C03649=1235.303,242.805,-59.932,-176.879,6.176,148.185
C03650=1235.299,243.053,-59.959,-176.877,6.178,148.185
C03651=1235.294,243.302,-59.985,-176.875,6.180,148.185
C03652=1235.290,243.551,-60.011,-176.872,6.182,148.184
C03653=1235.286,243.800,-60.036,-176.870,6.184,148.184
C03654=1235.281,244.047,-60.063,-176.867,6.186,148.184
C03655=1235.276,244.296,-60.089,-176.864,6.187,148.184
C03656=1235.272,244.545,-60.115,-176.862,6.189,148.183
C03657=1235.268,244.793,-60.141,-176.860,6.191,148.183
C03658=1235.263,245.043,-60.167,-176.858,6.193,148.183
C03659=1235.259,245.291,-60.193,-176.855,6.195,148.183
C03660=1235.254,245.539,-60.220,-176.852,6.196,148.182
C03661=1235.249,245.788,-60.246,-176.850,6.198,148.182
C03662=1235.246,246.036,-60.272,-176.847,6.200,148.182
C03663=1235.241,246.285,-60.298,-176.844,6.202,148.181
C03664=1235.236,246.534,-60.324,-176.842,6.204,148.181
C03665=1235.232,246.783,-60.351,-176.840,6.206,148.181
C03666=1235.227,247.031,-60.377,-176.837,6.208,148.181
C03667=1235.224,247.280,-60.404,-176.835,6.210,148.180
C03668=1235.218,247.528,-60.429,-176.832,6.211,148.180
C03669=1235.214,247.776,-60.456,-176.830,6.213,148.180
C03670=1235.209,248.025,-60.482,-176.828,6.215,148.180
C03671=1235.205,248.273,-60.509,-176.825,6.217,148.179
C03672=1235.200,248.523,-60.535,-176.823,6.219,148.179
C03673=1235.196,248.771,-60.562,-176.820,6.221,148.179
C03674=1235.192,249.020,-60.587,-176.817,6.223,148.178
C03675=1235.187,249.268,-60.614,-176.815,6.225,148.178
C03676=1235.183,249.517,-60.640,-176.813,6.227,148.178
C03677=1235.179,249.765,-60.667,-176.810,6.229,148.178
C03678=1235.175,250.013,-60.694,-176.807,6.231,148.177
C03679=1235.170,250.263,-60.720,-176.805,6.232,148.177
C03680=1235.166,250.511,-60.746,-176.802,6.234,148.177
C03681=1235.160,250.759,-60.772,-176.800,6.237,148.177
C03682=1235.156,251.007,-60.799,-176.797,6.238,148.176
C03683=1235.152,251.256,-60.826,-176.795,6.240,148.176
C03684=1235.147,251.505,-60.852,-176.793,6.241,148.176
C03685=1235.143,251.753,-60.879,-176.790,6.243,148.175
C03686=1235.138,252.002,-60.905,-176.788,6.245,148.175
C03687=1235.134,252.250,-60.932,-176.785,6.247,148.175
C03688=1235.129,252.499,-60.959,-176.783,6.249,148.175
C03689=1235.125,252.747,-60.985,-176.780,6.251,148.174
C03690=1235.120,252.996,-61.011,-176.778,6.253,148.174
C03691=1235.116,253.245,-61.039,-176.776,6.255,148.174
C03692=1235.112,253.493,-61.065,-176.773,6.257,148.174
C03693=1235.107,253.742,-61.091,-176.770,6.259,148.173
C03694=1235.103,253.990,-61.118,-176.768,6.261,148.173
C03695=1235.098,254.239,-61.145,-176.766,6.263,148.173
C03696=1235.093,254.487,-61.172,-176.763,6.265,148.173
C03697=1235.089,254.736,-61.198,-176.760,6.267,148.172
C03698=1235.085,254.985,-61.225,-176.758,6.269,148.172
C03699=1235.080,255.233,-61.252,-176.755,6.271,148.172
C03700=1235.076,255.481,-61.278,-176.753,6.273,148.172
C03701=1235.071,255.730,-61.305,-176.750,6.275,148.171
C03702=1235.067,255.978,-61.332,-176.748,6.277,148.171
C03703=1235.062,256.227,-61.358,-176.745,6.279,148.171
C03704=1235.058,256.476,-61.386,-176.743,6.281,148.171
C03705=1235.054,256.725,-61.413,-176.741,6.283,148.170
C03706=1235.050,256.973,-61.439,-176.738,6.285,148.170
C03707=1235.045,257.221,-61.466,-176.735,6.287,148.170
C03708=1235.041,257.470,-61.493,-176.733,6.289,148.170
C03709=1235.037,257.718,-61.520,-176.731,6.291,148.169
C03710=1235.032,257.967,-61.547,-176.728,6.293,148.169
C03711=1235.027,258.216,-61.573,-176.726,6.295,148.169
C03712=1235.022,258.464,-61.600,-176.723,6.297,148.169
C03713=1235.018,258.712,-61.627,-176.721,6.299,148.168
C03714=1235.014,258.961,-61.654,-176.718,6.300,148.168
C03715=1235.009,259.209,-61.681,-176.716,6.303,148.168
C03716=1235.004,259.458,-61.708,-176.713,6.305,148.168
C03717=1235.001,259.707,-61.735,-176.711,6.306,148.167
C03718=1234.996,259.955,-61.762,-176.708,6.308,148.167
C03719=1234.992,260.204,-61.789,-176.706,6.311,148.167
C03720=1234.987,260.452,-61.816,-176.703,6.312,148.167
C03721=1234.983,260.701,-61.843,-176.701,6.314,148.166
C03722=1234.979,260.949,-61.869,-176.699,6.317,148.166
C03723=1234.974,261.197,-61.897,-176.696,6.318,148.166
C03724=1234.970,261.445,-61.924,-176.694,6.320,148.166
C03725=1234.966,261.694,-61.952,-176.691,6.322,148.165
C03726=1234.961,261.943,-61.979,-176.689,6.324,148.165
C03727=1234.956,262.191,-62.006,-176.686,6.326,148.165
C03728=1234.952,262.440,-62.032,-176.684,6.328,148.165
C03729=1234.948,262.688,-62.059,-176.681,6.330,148.165
C03730=1234.943,262.937,-62.086,-176.679,6.332,148.164
C03731=1234.939,263.186,-62.114,-176.676,6.334,148.164
C03732=1234.934,263.458,-62.143,-176.674,6.336,148.164
C03733=1234.929,263.731,-62.174,-176.672,6.338,148.164
C03734=1234.925,264.003,-62.204,-176.668,6.341,148.163
C03735=1234.919,264.276,-62.234,-176.666,6.343,148.163
C03736=1234.915,264.524,-62.261,-176.663,6.345,148.163
C03737=1234.911,264.772,-62.287,-176.661,6.347,148.163
C03738=1234.906,265.021,-62.314,-176.659,6.349,148.162
C03739=1234.902,265.269,-62.343,-176.656,6.351,148.162
C03740=1234.898,265.518,-62.370,-176.654,6.353,148.162
C03741=1234.893,265.766,-62.397,-176.651,6.355,148.162
C03742=1234.888,266.015,-62.424,-176.649,6.357,148.161
C03743=1234.884,266.263,-62.452,-176.646,6.359,148.161
C03744=1234.880,266.512,-62.479,-176.644,6.361,148.161
C03745=1234.875,266.761,-62.506,-176.641,6.363,148.161
C03746=1234.871,267.009,-62.533,-176.639,6.365,148.161
C03747=1234.866,267.257,-62.561,-176.637,6.367,148.160
C03748=1234.862,267.506,-62.588,-176.634,6.369,148.160
C03749=1234.858,267.754,-62.616,-176.632,6.371,148.160
C03750=1234.853,268.002,-62.643,-176.629,6.373,148.160
C03751=1234.849,268.251,-62.670,-176.627,6.375,148.160
C03752=1234.845,268.500,-62.698,-176.625,6.377,148.159
C03753=1234.840,268.748,-62.725,-176.622,6.379,148.159
C03754=1234.836,268.997,-62.752,-176.619,6.382,148.159
C03755=1234.831,269.244,-62.780,-176.617,6.384,148.159
C03756=1234.827,269.494,-62.808,-176.614,6.386,148.159
C03757=1234.823,269.741,-62.835,-176.612,6.388,148.158
C03758=1234.817,269.990,-62.863,-176.609,6.390,148.158
C03759=1234.814,270.239,-62.891,-176.607,6.392,148.158
C03760=1234.809,270.487,-62.918,-176.605,6.394,148.158
C03761=1234.805,270.735,-62.946,-176.602,6.396,148.157
C03762=1234.800,270.984,-62.973,-176.600,6.398,148.157
C03763=1234.796,271.232,-63.001,-176.597,6.400,148.157
C03764=1234.792,271.481,-63.028,-176.595,6.402,148.157
C03765=1234.787,271.729,-63.056,-176.593,6.404,148.157
C03766=1234.783,271.978,-63.084,-176.590,6.406,148.156
C03767=1234.778,272.226,-63.112,-176.588,6.408,148.156
C03768=1234.773,272.475,-63.139,-176.585,6.410,148.156
C03769=1234.770,272.723,-63.167,-176.583,6.413,148.156
C03770=1234.765,272.972,-63.194,-176.581,6.414,148.156
C03771=1234.761,273.219,-63.222,-176.578,6.418,148.156
C03772=1234.757,273.468,-63.250,-176.575,6.419,148.155
C03773=1234.752,273.717,-63.278,-176.573,6.421,148.155
C03774=1234.747,273.965,-63.306,-176.571,6.424,148.155
C03775=1234.743,274.214,-63.333,-176.568,6.425,148.155
C03776=1234.739,274.462,-63.361,-176.566,6.428,148.155
C03777=1234.735,274.710,-63.389,-176.563,6.430,148.154
C03778=1234.730,274.959,-63.417,-176.561,6.432,148.154
C03779=1234.725,275.207,-63.444,-176.559,6.434,148.154
C03780=1234.722,275.456,-63.472,-176.556,6.436,148.154
C03781=1234.717,275.704,-63.500,-176.554,6.438,148.154
C03782=1234.712,275.952,-63.528,-176.551,6.440,148.153
C03783=1234.708,276.201,-63.556,-176.549,6.442,148.153
C03784=1234.704,276.449,-63.584,-176.546,6.445,148.153
C03785=1234.700,276.698,-63.611,-176.544,6.447,148.153
C03786=1234.695,276.946,-63.640,-176.541,6.449,148.153
C03787=1234.690,277.194,-63.667,-176.539,6.451,148.153
C03788=1234.686,277.443,-63.696,-176.537,6.453,148.152
C03789=1234.682,277.690,-63.723,-176.535,6.455,148.152
C03790=1234.677,277.940,-63.751,-176.532,6.457,148.152
C03791=1234.673,278.188,-63.779,-176.530,6.459,148.152
C03792=1234.669,278.436,-63.807,-176.527,6.461,148.152
C03793=1234.664,278.685,-63.836,-176.525,6.463,148.152
C03794=1234.660,278.933,-63.864,-176.523,6.465,148.151
C03795=1234.656,279.181,-63.892,-176.520,6.468,148.151
C03796=1234.651,279.430,-63.919,-176.517,6.470,148.151
C03797=1234.647,279.678,-63.947,-176.515,6.473,148.151
C03798=1234.642,279.927,-63.976,-176.513,6.474,148.151
C03799=1234.638,280.175,-64.004,-176.511,6.477,148.151
C03800=1234.634,280.423,-64.032,-176.508,6.479,148.150
C03801=1234.629,280.672,-64.060,-176.506,6.481,148.150
C03802=1234.625,280.920,-64.088,-176.503,6.483,148.150
C03803=1234.621,281.168,-64.116,-176.501,6.485,148.150
C03804=1234.616,281.417,-64.145,-176.498,6.488,148.150
C03805=1234.612,281.665,-64.173,-176.496,6.490,148.150
C03806=1234.607,281.913,-64.201,-176.493,6.492,148.149
C03807=1234.603,282.162,-64.229,-176.491,6.494,148.149
C03808=1234.598,282.410,-64.258,-176.489,6.496,148.149
C03809=1234.595,282.659,-64.286,-176.487,6.498,148.149
C03810=1234.590,282.907,-64.314,-176.484,6.500,148.149
C03811=1234.586,283.156,-64.342,-176.482,6.502,148.148
C03812=1234.581,283.403,-64.370,-176.480,6.504,148.148
C03813=1234.577,283.652,-64.399,-176.477,6.507,148.148
C03814=1234.573,283.900,-64.427,-176.475,6.509,148.148
C03815=1234.568,284.149,-64.455,-176.472,6.511,148.148
C03816=1234.564,284.397,-64.483,-176.470,6.514,148.148
C03817=1234.559,284.646,-64.512,-176.468,6.516,148.148
C03818=1234.555,284.894,-64.540,-176.465,6.518,148.147
C03819=1234.551,285.142,-64.569,-176.463,6.520,148.147
C03820=1234.547,285.391,-64.597,-176.460,6.523,148.147
C03821=1234.542,285.639,-64.626,-176.458,6.525,148.147
C03822=1234.538,285.887,-64.654,-176.455,6.527,148.147
C03823=1234.533,286.135,-64.682,-176.453,6.529,148.147
C03824=1234.529,286.384,-64.711,-176.451,6.531,148.147
C03825=1234.524,286.632,-64.739,-176.448,6.533,148.146
C03826=1234.520,286.881,-64.768,-176.446,6.535,148.146
C03827=1234.516,287.129,-64.796,-176.444,6.537,148.146
C03828=1234.511,287.377,-64.825,-176.441,6.540,148.146
C03829=1234.507,287.626,-64.853,-176.439,6.543,148.146
C03830=1234.503,287.873,-64.882,-176.436,6.544,148.146
C03831=1234.498,288.122,-64.911,-176.434,6.547,148.146
C03832=1234.494,288.371,-64.939,-176.432,6.549,148.146
C03833=1234.489,288.619,-64.967,-176.430,6.551,148.145
C03834=1234.485,288.867,-64.997,-176.427,6.554,148.145
C03835=1234.481,289.116,-65.025,-176.424,6.556,148.145
C03836=1234.476,289.390,-65.056,-176.422,6.558,148.145
C03837=1234.471,289.664,-65.088,-176.419,6.561,148.145
C03838=1234.467,289.938,-65.120,-176.417,6.563,148.145
C03839=1234.461,290.211,-65.151,-176.414,6.566,148.144
C03840=1234.458,290.460,-65.179,-176.412,6.568,148.144
C03841=1234.453,290.708,-65.209,-176.410,6.570,148.144
C03842=1234.448,290.956,-65.237,-176.407,6.572,148.144
C03843=1234.444,291.205,-65.265,-176.405,6.574,148.144
C03844=1234.440,291.453,-65.295,-176.403,6.577,148.144
C03845=1234.435,291.701,-65.323,-176.400,6.579,148.144
C03846=1234.432,291.949,-65.352,-176.398,6.582,148.144
C03847=1234.427,292.198,-65.381,-176.395,6.584,148.143
C03848=1234.422,292.446,-65.409,-176.393,6.586,148.143
C03849=1234.418,292.695,-65.439,-176.391,6.588,148.143
C03850=1234.414,292.943,-65.467,-176.389,6.590,148.143
C03851=1234.410,293.192,-65.496,-176.386,6.593,148.143
C03852=1234.405,293.440,-65.525,-176.383,6.595,148.143
C03853=1234.401,293.688,-65.554,-176.381,6.597,148.143
C03854=1234.397,293.937,-65.582,-176.379,6.600,148.143
C03855=1234.392,294.184,-65.611,-176.377,6.601,148.142
C03856=1234.388,294.433,-65.640,-176.375,6.604,148.142
C03857=1234.384,294.681,-65.669,-176.372,6.607,148.142
C03858=1234.379,294.930,-65.699,-176.370,6.609,148.142
C03859=1234.375,295.177,-65.727,-176.367,6.611,148.142
C03860=1234.371,295.426,-65.756,-176.365,6.613,148.142
C03861=1234.366,295.675,-65.785,-176.363,6.615,148.142
C03862=1234.362,295.923,-65.814,-176.361,6.618,148.142
C03863=1234.357,296.170,-65.843,-176.358,6.620,148.142
C03864=1234.353,296.419,-65.872,-176.356,6.623,148.142
C03865=1234.350,296.667,-65.901,-176.354,6.625,148.141
C03866=1234.345,296.916,-65.930,-176.351,6.627,148.141
C03867=1234.340,297.164,-65.959,-176.349,6.629,148.141
C03868=1234.336,297.412,-65.988,-176.346,6.632,148.141
C03869=1234.332,297.660,-66.018,-176.344,6.634,148.141
C03870=1234.327,297.909,-66.046,-176.342,6.636,148.141
C03871=1234.323,298.157,-66.076,-176.339,6.638,148.141
C03872=1234.318,298.405,-66.105,-176.337,6.641,148.141
C03873=1234.314,298.654,-66.134,-176.335,6.643,148.141
C03874=1234.310,298.902,-66.163,-176.333,6.646,148.141
C03875=1234.306,299.150,-66.192,-176.331,6.648,148.141
C03876=1234.302,299.398,-66.221,-176.328,6.650,148.140
C03877=1234.297,299.647,-66.250,-176.326,6.652,148.140
C03878=1234.293,299.895,-66.279,-176.324,6.654,148.140
C03879=1234.289,300.143,-66.309,-176.321,6.657,148.140
C03880=1234.284,300.391,-66.338,-176.319,6.660,148.140
C03881=1234.280,300.639,-66.367,-176.317,6.662,148.140
C03882=1234.276,300.887,-66.397,-176.314,6.664,148.140
C03883=1234.271,301.136,-66.426,-176.312,6.666,148.140
C03884=1234.267,301.384,-66.455,-176.310,6.669,148.140
C03885=1234.263,301.633,-66.484,-176.307,6.671,148.140
C03886=1234.259,301.881,-66.514,-176.305,6.674,148.140
C03887=1234.254,302.129,-66.543,-176.303,6.676,148.140
C03888=1234.250,302.377,-66.572,-176.301,6.678,148.139
C03889=1234.245,302.625,-66.602,-176.298,6.681,148.139
C03890=1234.241,302.873,-66.631,-176.296,6.683,148.139
C03891=1234.237,303.122,-66.660,-176.294,6.685,148.139
C03892=1234.233,303.370,-66.690,-176.292,6.687,148.139
C03893=1234.228,303.619,-66.719,-176.290,6.690,148.139
C03894=1234.224,303.867,-66.748,-176.287,6.693,148.139
C03895=1234.219,304.114,-66.778,-176.285,6.695,148.139
C03896=1234.214,304.363,-66.808,-176.282,6.697,148.139
C03897=1234.210,304.611,-66.837,-176.280,6.699,148.139
C03898=1234.206,304.860,-66.866,-176.278,6.701,148.139
C03899=1234.202,305.108,-66.896,-176.275,6.704,148.139
C03900=1234.198,305.356,-66.925,-176.273,6.707,148.139
C03901=1234.194,305.604,-66.955,-176.271,6.709,148.139
C03902=1234.189,305.853,-66.984,-176.269,6.711,148.138
C03903=1234.185,306.100,-67.014,-176.266,6.714,148.138
C03904=1234.181,306.349,-67.044,-176.264,6.716,148.138
C03905=1234.176,306.597,-67.074,-176.262,6.719,148.138
C03906=1234.172,306.845,-67.103,-176.260,6.721,148.138
C03907=1234.167,307.093,-67.133,-176.258,6.723,148.138
C03908=1234.163,307.341,-67.162,-176.255,6.726,148.138
C03909=1234.159,307.589,-67.191,-176.253,6.728,148.138
C03910=1234.155,307.838,-67.221,-176.251,6.730,148.138
C03911=1234.150,308.086,-67.251,-176.249,6.733,148.138
C03912=1234.146,308.334,-67.281,-176.247,6.735,148.138
C03913=1234.142,308.582,-67.311,-176.244,6.738,148.138
C03914=1234.138,308.831,-67.340,-176.242,6.740,148.138
C03915=1234.134,309.079,-67.369,-176.240,6.742,148.138
C03916=1234.129,309.327,-67.399,-176.238,6.744,148.138
C03917=1234.125,309.575,-67.430,-176.235,6.748,148.138
C03918=1234.121,309.823,-67.459,-176.233,6.750,148.138
C03919=1234.116,310.072,-67.489,-176.231,6.752,148.138
C03920=1234.111,310.320,-67.519,-176.229,6.754,148.138
C03921=1234.108,310.568,-67.549,-176.227,6.756,148.137
C03922=1234.103,310.816,-67.578,-176.224,6.760,148.137
C03923=1234.099,311.064,-67.608,-176.222,6.762,148.137
C03924=1234.094,311.313,-67.638,-176.220,6.764,148.137
C03925=1234.090,311.561,-67.668,-176.218,6.766,148.137
C03926=1234.086,311.809,-67.697,-176.215,6.769,148.137
C03927=1234.081,312.057,-67.727,-176.213,6.772,148.137
C03928=1234.077,312.305,-67.758,-176.211,6.774,148.137
C03929=1234.073,312.553,-67.787,-176.209,6.776,148.137
C03930=1234.068,312.802,-67.817,-176.206,6.779,148.137
C03931=1234.064,313.050,-67.847,-176.204,6.781,148.137
C03932=1234.060,313.298,-67.877,-176.202,6.784,148.137
C03933=1234.056,313.546,-67.907,-176.200,6.786,148.137
C03934=1234.051,313.794,-67.937,-176.198,6.788,148.137
C03935=1234.047,314.042,-67.966,-176.195,6.791,148.137
C03936=1234.043,314.291,-67.998,-176.193,6.794,148.137
C03937=1234.039,314.539,-68.027,-176.191,6.796,148.137
C03938=1234.035,314.787,-68.057,-176.189,6.798,148.137
C03939=1234.030,315.035,-68.087,-176.187,6.801,148.137
C03940=1234.026,315.310,-68.120,-176.184,6.803,148.137
C03941=1234.021,315.587,-68.154,-176.182,6.806,148.137
C03942=1234.017,315.862,-68.188,-176.180,6.809,148.137
C03943=1234.012,316.137,-68.220,-176.177,6.812,148.137
C03944=1234.007,316.385,-68.251,-176.175,6.814,148.137
C03945=1234.003,316.634,-68.281,-176.173,6.816,148.137
C03946=1233.998,316.882,-68.311,-176.171,6.819,148.137
C03947=1233.995,317.131,-68.341,-176.169,6.822,148.137
C03948=1233.990,317.379,-68.372,-176.167,6.824,148.137
C03949=1233.986,317.627,-68.401,-176.164,6.826,148.137
C03950=1233.981,317.875,-68.432,-176.162,6.829,148.137
C03951=1233.977,318.122,-68.462,-176.160,6.831,148.137
C03952=1233.972,318.371,-68.492,-176.158,6.834,148.137
C03953=1233.969,318.619,-68.523,-176.156,6.836,148.137
C03954=1233.964,318.867,-68.553,-176.153,6.839,148.137
C03955=1233.960,319.116,-68.583,-176.151,6.842,148.137
C03956=1233.956,319.364,-68.614,-176.149,6.844,148.137
C03957=1233.952,319.612,-68.643,-176.147,6.846,148.137
C03958=1233.947,319.860,-68.674,-176.145,6.849,148.137
C03959=1233.943,320.107,-68.704,-176.143,6.852,148.137
C03960=1233.938,320.355,-68.735,-176.141,6.854,148.137
C03961=1233.935,320.604,-68.765,-176.139,6.856,148.137
C03962=1233.930,320.852,-68.796,-176.136,6.858,148.137
C03963=1233.926,321.100,-68.826,-176.134,6.862,148.137
C03964=1233.921,321.349,-68.856,-176.132,6.864,148.137
C03965=1233.917,321.597,-68.887,-176.130,6.866,148.137
C03966=1233.913,321.844,-68.917,-176.128,6.868,148.137
C03967=1233.909,322.093,-68.948,-176.126,6.872,148.137
C03968=1233.905,322.340,-68.978,-176.124,6.874,148.137
C03969=1233.900,322.589,-69.008,-176.122,6.876,148.137
C03970=1233.896,322.837,-69.039,-176.120,6.878,148.137
C03971=1233.892,323.085,-69.069,-176.117,6.882,148.137
C03972=1233.888,323.333,-69.100,-176.115,6.884,148.137
C03973=1233.884,323.581,-69.130,-176.113,6.886,148.137
C03974=1233.879,323.830,-69.160,-176.111,6.888,148.137
C03975=1233.874,324.077,-69.191,-176.110,6.891,148.137
C03976=1233.871,324.326,-69.222,-176.107,6.894,148.137
C03977=1233.866,324.574,-69.252,-176.105,6.896,148.137
C03978=1233.862,324.822,-69.283,-176.103,6.899,148.138
C03979=1233.858,325.069,-69.313,-176.101,6.901,148.138
C03980=1233.854,325.318,-69.344,-176.098,6.904,148.138
C03981=1233.849,325.566,-69.375,-176.097,6.907,148.138
C03982=1233.845,325.814,-69.405,-176.095,6.909,148.138
C03983=1233.841,326.062,-69.436,-176.093,6.911,148.138
C03984=1233.837,326.310,-69.467,-176.090,6.915,148.138
C03985=1233.832,326.558,-69.498,-176.088,6.917,148.138
C03986=1233.828,326.806,-69.528,-176.086,6.919,148.138
C03987=1233.824,327.055,-69.559,-176.085,6.922,148.138
C03988=1233.820,327.303,-69.590,-176.082,6.925,148.138
C03989=1233.816,327.550,-69.620,-176.080,6.927,148.138
C03990=1233.811,327.798,-69.651,-176.078,6.929,148.138
C03991=1233.807,328.047,-69.682,-176.076,6.932,148.138
C03992=1233.803,328.295,-69.713,-176.075,6.934,148.138
C03993=1233.799,328.542,-69.743,-176.072,6.937,148.138
C03994=1233.795,328.791,-69.774,-176.070,6.939,148.138
C03995=1233.790,329.039,-69.805,-176.068,6.942,148.138
C03996=1233.785,329.287,-69.836,-176.066,6.944,148.138
C03997=1233.781,329.536,-69.867,-176.064,6.948,148.139
C03998=1233.778,329.783,-69.897,-176.062,6.950,148.139
C03999=1233.773,330.031,-69.928,-176.060,6.952,148.138
C04000=1233.769,330.280,-69.959,-176.058,6.955,148.139
C04001=1233.765,330.527,-69.990,-176.056,6.958,148.139
C04002=1233.760,330.775,-70.021,-176.054,6.960,148.139
C04003=1233.756,331.024,-70.052,-176.052,6.962,148.139
C04004=1233.752,331.271,-70.083,-176.050,6.965,148.139
C04005=1233.747,331.519,-70.113,-176.048,6.967,148.139
C04006=1233.744,331.767,-70.145,-176.046,6.971,148.139
C04007=1233.739,332.015,-70.176,-176.044,6.973,148.139
C04008=1233.735,332.263,-70.207,-176.042,6.975,148.139
C04009=1233.731,332.512,-70.238,-176.040,6.978,148.139
C04010=1233.726,332.760,-70.269,-176.038,6.981,148.140
C04011=1233.722,333.007,-70.300,-176.036,6.983,148.139
C04012=1233.718,333.256,-70.331,-176.034,6.986,148.140
C04013=1233.714,333.504,-70.361,-176.032,6.988,148.140
C04014=1233.710,333.752,-70.392,-176.030,6.991,148.140
C04015=1233.705,334.000,-70.424,-176.028,6.993,148.140
C04016=1233.701,334.248,-70.455,-176.026,6.996,148.140
C04017=1233.697,334.496,-70.486,-176.024,6.998,148.140
C04018=1233.692,334.744,-70.517,-176.023,7.001,148.140
C04019=1233.688,334.992,-70.548,-176.020,7.004,148.140
C04020=1233.684,335.240,-70.579,-176.018,7.006,148.140
C04021=1233.680,335.488,-70.611,-176.016,7.009,148.140
C04022=1233.676,335.736,-70.642,-176.015,7.011,148.140
C04023=1233.671,335.984,-70.673,-176.013,7.014,148.141
C04024=1233.667,336.232,-70.704,-176.010,7.017,148.141
C04025=1233.663,336.480,-70.735,-176.009,7.019,148.141
C04026=1233.659,336.728,-70.767,-176.007,7.022,148.141
C04027=1233.654,336.976,-70.798,-176.005,7.024,148.141
C04028=1233.650,337.223,-70.829,-176.003,7.027,148.141
C04029=1233.646,337.472,-70.860,-176.001,7.030,148.141
C04030=1233.641,337.720,-70.891,-175.999,7.032,148.141
C04031=1233.638,337.968,-70.923,-175.997,7.034,148.141
C04032=1233.633,338.216,-70.954,-175.995,7.037,148.141
C04033=1233.629,338.464,-70.986,-175.993,7.040,148.142
C04034=1233.625,338.712,-71.016,-175.991,7.043,148.142
C04035=1233.621,338.960,-71.048,-175.990,7.045,148.142
C04036=1233.616,339.208,-71.079,-175.988,7.048,148.142
C04037=1233.613,339.456,-71.111,-175.986,7.050,148.142
C04038=1233.608,339.703,-71.142,-175.984,7.053,148.142
C04039=1233.604,339.952,-71.173,-175.982,7.056,148.142
C04040=1233.599,340.200,-71.206,-175.980,7.058,148.142
C04041=1233.595,340.448,-71.237,-175.978,7.061,148.143
C04042=1233.591,340.696,-71.268,-175.977,7.063,148.143
C04043=1233.587,340.944,-71.299,-175.975,7.066,148.143
C04044=1233.582,341.221,-71.335,-175.972,7.069,148.143
C04045=1233.578,341.499,-71.370,-175.970,7.072,148.143
C04046=1233.573,341.776,-71.405,-175.969,7.075,148.143
C04047=1233.568,342.054,-71.440,-175.966,7.078,148.143
C04048=1233.564,342.302,-71.471,-175.964,7.080,148.144
C04049=1233.560,342.550,-71.503,-175.963,7.083,148.144
C04050=1233.555,342.798,-71.535,-175.961,7.086,148.144
C04051=1233.551,343.046,-71.566,-175.959,7.088,148.144
C04052=1233.547,343.294,-71.598,-175.957,7.091,148.144
C04053=1233.543,343.541,-71.629,-175.955,7.093,148.144
C04054=1233.539,343.789,-71.661,-175.954,7.096,148.144
C04055=1233.534,344.038,-71.693,-175.952,7.098,148.144
C04056=1233.530,344.286,-71.724,-175.949,7.102,148.145
C04057=1233.526,344.533,-71.756,-175.948,7.104,148.145
C04058=1233.522,344.781,-71.788,-175.946,7.107,148.145
C04059=1233.518,345.030,-71.819,-175.945,7.109,148.145
C04060=1233.513,345.277,-71.851,-175.942,7.111,148.145
C04061=1233.509,345.526,-71.883,-175.940,7.115,148.145
C04062=1233.505,345.773,-71.914,-175.939,7.117,148.146
C04063=1233.501,346.022,-71.945,-175.937,7.120,148.146
C04064=1233.496,346.269,-71.977,-175.935,7.122,148.146
C04065=1233.492,346.517,-72.009,-175.934,7.125,148.146
C04066=1233.488,346.765,-72.041,-175.932,7.127,148.146
C04067=1233.484,347.013,-72.073,-175.930,7.131,148.146
C04068=1233.480,347.261,-72.105,-175.928,7.133,148.147
C04069=1233.475,347.509,-72.136,-175.926,7.136,148.147
C04070=1233.471,347.757,-72.168,-175.925,7.138,148.147
C04071=1233.467,348.005,-72.200,-175.923,7.141,148.147
C04072=1233.463,348.253,-72.232,-175.921,7.143,148.147
C04073=1233.459,348.501,-72.263,-175.919,7.147,148.148
C04074=1233.455,348.749,-72.296,-175.918,7.149,148.148
C04075=1233.450,348.996,-72.327,-175.916,7.152,148.148
C04076=1233.447,349.244,-72.359,-175.914,7.154,148.148
C04077=1233.441,349.492,-72.391,-175.913,7.157,148.148
C04078=1233.438,349.740,-72.423,-175.911,7.159,148.148
C04079=1233.434,349.988,-72.455,-175.909,7.162,148.148
C04080=1233.429,350.236,-72.487,-175.907,7.165,148.149
C04081=1233.425,350.484,-72.519,-175.905,7.167,148.149
C04082=1233.422,350.732,-72.551,-175.904,7.170,148.149
C04083=1233.417,350.979,-72.583,-175.902,7.172,148.149
C04084=1233.413,351.228,-72.615,-175.900,7.175,148.149
C04085=1233.409,351.476,-72.647,-175.899,7.177,148.150
C04086=1233.404,351.723,-72.679,-175.897,7.181,148.150
C04087=1233.400,351.971,-72.710,-175.895,7.183,148.150
C04088=1233.396,352.220,-72.743,-175.893,7.186,148.150
C04089=1233.392,352.467,-72.774,-175.892,7.188,148.150
C04090=1233.387,352.715,-72.807,-175.890,7.191,148.151
C04091=1233.383,352.963,-72.839,-175.889,7.194,148.151
C04092=1233.379,353.211,-72.870,-175.887,7.196,148.151
C04093=1233.375,353.459,-72.903,-175.886,7.199,148.151
C04094=1233.371,353.707,-72.934,-175.884,7.202,148.152
C04095=1233.367,353.955,-72.967,-175.882,7.205,148.152
C04096=1233.363,354.202,-72.999,-175.880,7.207,148.152
C04097=1233.358,354.450,-73.032,-175.879,7.210,148.152
C04098=1233.354,354.699,-73.063,-175.877,7.212,148.152
C04099=1233.349,354.946,-73.095,-175.876,7.215,148.152
C04100=1233.346,355.194,-73.127,-175.874,7.217,148.153
C04101=1233.341,355.443,-73.160,-175.872,7.220,148.153
C04102=1233.338,355.690,-73.192,-175.871,7.223,148.153
C04103=1233.333,355.938,-73.224,-175.869,7.226,148.153
C04104=1233.329,356.186,-73.256,-175.867,7.229,148.154
C04105=1233.325,356.434,-73.289,-175.866,7.231,148.154
C04106=1233.321,356.682,-73.320,-175.864,7.234,148.154
C04107=1233.316,356.929,-73.353,-175.863,7.236,148.154
C04108=1233.312,357.177,-73.385,-175.861,7.239,148.154
C04109=1233.308,357.425,-73.418,-175.860,7.242,148.155
C04110=1233.305,357.673,-73.450,-175.858,7.244,148.155
C04111=1233.300,357.921,-73.482,-175.857,7.247,148.155
C04112=1233.296,358.169,-73.514,-175.855,7.249,148.155
C04113=1233.291,358.417,-73.546,-175.853,7.253,148.156
C04114=1233.287,358.665,-73.580,-175.851,7.255,148.156
C04115=1233.283,358.912,-73.611,-175.850,7.258,148.156
C04116=1233.279,359.160,-73.644,-175.848,7.261,148.156
C04117=1233.275,359.408,-73.676,-175.847,7.263,148.157
C04118=1233.271,359.656,-73.709,-175.845,7.266,148.157
C04119=1233.266,359.904,-73.741,-175.844,7.268,148.157
C04120=1233.262,360.151,-73.773,-175.842,7.271,148.157
C04121=1233.258,360.400,-73.806,-175.841,7.274,148.158
C04122=1233.254,360.647,-73.838,-175.839,7.276,148.158
C04123=1233.250,360.895,-73.871,-175.838,7.279,148.158
C04124=1233.246,361.144,-73.903,-175.836,7.281,148.158
C04125=1233.242,361.390,-73.935,-175.835,7.284,148.158
C04126=1233.237,361.639,-73.968,-175.834,7.287,148.159
C04127=1233.233,361.886,-74.001,-175.832,7.289,148.159
C04128=1233.229,362.134,-74.033,-175.830,7.292,148.159
C04129=1233.225,362.382,-74.066,-175.829,7.296,148.160
C04130=1233.221,362.631,-74.098,-175.827,7.298,148.160
C04131=1233.216,362.878,-74.130,-175.825,7.301,148.160
C04132=1233.212,363.126,-74.163,-175.824,7.303,148.160
C04133=1233.208,363.374,-74.195,-175.823,7.306,148.161
C04134=1233.204,363.621,-74.228,-175.821,7.308,148.161
C04135=1233.200,363.870,-74.260,-175.820,7.311,148.161
C04136=1233.196,364.117,-74.294,-175.818,7.314,148.161
C04137=1233.192,364.365,-74.327,-175.817,7.316,148.162
C04138=1233.187,364.613,-74.358,-175.815,7.319,148.162
C04139=1233.183,364.860,-74.391,-175.814,7.322,148.162
C04140=1233.179,365.109,-74.424,-175.813,7.325,148.163
C04141=1233.175,365.356,-74.456,-175.811,7.327,148.163
C04142=1233.171,365.604,-74.489,-175.809,7.330,148.163
C04143=1233.167,365.852,-74.522,-175.808,7.332,148.163
C04144=1233.162,366.100,-74.554,-175.807,7.335,148.164
C04145=1233.159,366.348,-74.587,-175.805,7.338,148.164
C04146=1233.154,366.595,-74.620,-175.804,7.340,148.164
C04147=1233.150,366.843,-74.652,-175.803,7.343,148.165
C04148=1233.145,367.123,-74.690,-175.801,7.346,148.165
C04149=1233.141,367.402,-74.727,-175.800,7.349,148.165
C04150=1233.136,367.682,-74.763,-175.798,7.352,148.165
C04151=1233.132,367.961,-74.800,-175.797,7.355,148.166
C04152=1233.128,368.209,-74.833,-175.795,7.357,148.166
C04153=1233.123,368.457,-74.866,-175.794,7.360,148.166
C04154=1233.119,368.705,-74.899,-175.792,7.363,148.167
C04155=1233.114,368.952,-74.932,-175.791,7.365,148.167
C04156=1233.110,369.200,-74.964,-175.790,7.368,148.167
C04157=1233.107,369.447,-74.997,-175.788,7.371,148.168
C04158=1233.102,369.695,-75.030,-175.787,7.374,148.168
C04159=1233.098,369.943,-75.063,-175.785,7.376,148.168
C04160=1233.094,370.191,-75.095,-175.784,7.379,148.169
C04161=1233.090,370.439,-75.128,-175.783,7.382,148.169
C04162=1233.086,370.687,-75.162,-175.782,7.384,148.169
C04163=1233.081,370.934,-75.195,-175.780,7.386,148.169
C04164=1233.078,371.183,-75.227,-175.779,7.389,148.170
C04165=1233.074,371.430,-75.260,-175.778,7.392,148.170
C04166=1233.070,371.678,-75.293,-175.777,7.394,148.170
C04167=1233.065,371.926,-75.326,-175.775,7.397,148.171
C04168=1233.061,372.173,-75.359,-175.774,7.400,148.171
C04169=1233.057,372.422,-75.392,-175.773,7.402,148.171
C04170=1233.053,372.670,-75.425,-175.771,7.405,148.172
C04171=1233.049,372.917,-75.458,-175.770,7.408,148.172
C04172=1233.044,373.165,-75.491,-175.769,7.410,148.172
C04173=1233.040,373.413,-75.524,-175.768,7.413,148.173
C04174=1233.037,373.660,-75.557,-175.766,7.415,148.173
C04175=1233.032,373.908,-75.589,-175.765,7.418,148.173
C04176=1233.028,374.156,-75.622,-175.764,7.421,148.174
C04177=1233.024,374.404,-75.656,-175.762,7.423,148.174
C04178=1233.020,374.652,-75.689,-175.761,7.426,148.174
C04179=1233.016,374.899,-75.722,-175.761,7.428,148.175
C04180=1233.012,375.147,-75.755,-175.760,7.431,148.175
C04181=1233.008,375.395,-75.788,-175.758,7.434,148.175
C04182=1233.003,375.643,-75.821,-175.757,7.436,148.176
C04183=1232.999,375.890,-75.855,-175.756,7.439,148.176
C04184=1232.995,376.138,-75.888,-175.754,7.442,148.176
C04185=1232.991,376.386,-75.921,-175.753,7.444,148.176
C04186=1232.987,376.633,-75.954,-175.752,7.447,148.177
C04187=1232.983,376.881,-75.987,-175.751,7.449,148.177
C04188=1232.979,377.129,-76.020,-175.750,7.452,148.178
C04189=1232.974,377.377,-76.053,-175.748,7.455,148.178
C04190=1232.970,377.624,-76.087,-175.748,7.457,148.178
C04191=1232.966,377.872,-76.120,-175.747,7.460,148.179
C04192=1232.962,378.120,-76.153,-175.745,7.462,148.179
C04193=1232.958,378.368,-76.186,-175.744,7.465,148.179
C04194=1232.954,378.615,-76.219,-175.743,7.468,148.180
C04195=1232.950,378.863,-76.252,-175.742,7.470,148.180
C04196=1232.945,379.111,-76.286,-175.741,7.473,148.180
C04197=1232.941,379.358,-76.319,-175.740,7.475,148.181
C04198=1232.937,379.606,-76.352,-175.738,7.478,148.181
C04199=1232.933,379.854,-76.385,-175.737,7.480,148.181
C04200=1232.929,380.102,-76.418,-175.736,7.483,148.182
C04201=1232.924,380.350,-76.452,-175.735,7.486,148.182
C04202=1232.920,380.597,-76.485,-175.734,7.488,148.182
C04203=1232.916,380.845,-76.518,-175.733,7.490,148.183
C04204=1232.912,381.093,-76.551,-175.732,7.493,148.183
C04205=1232.908,381.341,-76.586,-175.731,7.496,148.183
C04206=1232.904,381.588,-76.619,-175.729,7.498,148.184
C04207=1232.900,381.836,-76.652,-175.729,7.500,148.184
C04208=1232.896,382.084,-76.685,-175.728,7.503,148.185
C04209=1232.892,382.332,-76.718,-175.726,7.506,148.185
C04210=1232.888,382.579,-76.751,-175.726,7.508,148.185
C04211=1232.883,382.827,-76.785,-175.725,7.511,148.186
C04212=1232.879,383.075,-76.819,-175.723,7.514,148.186
C04213=1232.875,383.322,-76.852,-175.722,7.517,148.187
C04214=1232.871,383.570,-76.885,-175.721,7.518,148.187
C04215=1232.867,383.818,-76.919,-175.720,7.521,148.187
C04216=1232.863,384.066,-76.952,-175.719,7.524,148.187
C04217=1232.859,384.313,-76.986,-175.718,7.526,148.188
C04218=1232.854,384.561,-77.020,-175.717,7.529,148.188
C04219=1232.850,384.809,-77.053,-175.716,7.532,148.189
C04220=1232.846,385.057,-77.086,-175.715,7.534,148.189
C04221=1232.842,385.304,-77.120,-175.714,7.536,148.189
C04222=1232.838,385.552,-77.153,-175.713,7.539,148.190
C04223=1232.834,385.799,-77.186,-175.712,7.541,148.190
C04224=1232.830,386.048,-77.220,-175.711,7.544,148.190
C04225=1232.826,386.295,-77.254,-175.710,7.547,148.191
C04226=1232.822,386.543,-77.287,-175.709,7.549,148.191
C04227=1232.818,386.791,-77.320,-175.708,7.552,148.192
C04228=1232.814,387.038,-77.354,-175.708,7.554,148.192
C04229=1232.809,387.286,-77.388,-175.707,7.556,148.192
C04230=1232.805,387.533,-77.421,-175.705,7.559,148.193
C04231=1232.802,387.781,-77.455,-175.705,7.561,148.193
C04232=1232.797,388.029,-77.489,-175.704,7.564,148.194
C04233=1232.792,388.277,-77.522,-175.703,7.566,148.194
C04234=1232.789,388.524,-77.556,-175.702,7.569,148.194
C04235=1232.785,388.772,-77.589,-175.701,7.572,148.195
C04236=1232.780,389.020,-77.623,-175.700,7.574,148.195
C04237=1232.777,389.267,-77.657,-175.699,7.577,148.195
C04238=1232.772,389.515,-77.691,-175.698,7.579,148.196
C04239=1232.768,389.763,-77.724,-175.697,7.581,148.196
C04240=1232.764,390.010,-77.758,-175.696,7.584,148.197
C04241=1232.759,390.258,-77.791,-175.695,7.586,148.197
C04242=1232.756,390.505,-77.825,-175.694,7.589,148.197
C04243=1232.752,390.754,-77.859,-175.694,7.591,148.198
C04244=1232.748,391.002,-77.892,-175.692,7.594,148.198
C04245=1232.743,391.249,-77.926,-175.692,7.596,148.198
C04246=1232.739,391.497,-77.959,-175.691,7.599,148.199
C04247=1232.735,391.744,-77.993,-175.690,7.601,148.199
C04248=1232.732,391.992,-78.027,-175.689,7.603,148.200
C04249=1232.727,392.240,-78.061,-175.688,7.605,148.200
C04250=1232.723,392.487,-78.095,-175.687,7.609,148.200
C04251=1232.719,392.735,-78.128,-175.686,7.611,148.201
C04252=1232.715,393.017,-78.167,-175.686,7.613,148.201
C04253=1232.710,393.297,-78.205,-175.685,7.616,148.202
C04254=1232.704,393.579,-78.243,-175.683,7.619,148.202
C04255=1232.700,393.860,-78.282,-175.683,7.622,148.203
C04256=1232.696,394.108,-78.315,-175.682,7.624,148.203
C04257=1232.692,394.355,-78.349,-175.681,7.627,148.203
C04258=1232.688,394.604,-78.383,-175.680,7.629,148.204
C04259=1232.684,394.851,-78.417,-175.679,7.632,148.204
C04260=1232.680,395.098,-78.450,-175.678,7.634,148.204
C04261=1232.675,395.346,-78.485,-175.677,7.637,148.205
C04262=1232.672,395.594,-78.519,-175.677,7.638,148.205
C04263=1232.668,395.841,-78.552,-175.676,7.641,148.206
C04264=1232.663,396.089,-78.587,-175.675,7.644,148.206
C04265=1232.659,396.337,-78.620,-175.674,7.646,148.207
C04266=1232.655,396.584,-78.654,-175.674,7.648,148.207
C04267=1232.651,396.832,-78.688,-175.673,7.650,148.207
C04268=1232.647,397.079,-78.722,-175.672,7.653,148.208
C04269=1232.643,397.327,-78.756,-175.671,7.655,148.208
C04270=1232.639,397.575,-78.789,-175.670,7.658,148.208
C04271=1232.635,397.823,-78.824,-175.670,7.660,148.209
C04272=1232.631,398.070,-78.857,-175.669,7.663,148.209
C04273=1232.627,398.318,-78.891,-175.668,7.665,148.210
C04274=1232.623,398.566,-78.926,-175.667,7.667,148.210
C04275=1232.619,398.813,-78.959,-175.666,7.670,148.210
C04276=1232.614,399.061,-78.994,-175.666,7.672,148.211
C04277=1232.610,399.308,-79.028,-175.664,7.675,148.211
C04278=1232.607,399.556,-79.061,-175.664,7.677,148.212
C04279=1232.602,399.804,-79.096,-175.664,7.679,148.212
C04280=1232.598,400.051,-79.129,-175.663,7.682,148.212
C04281=1232.593,400.299,-79.163,-175.662,7.684,148.213
C04282=1232.590,400.547,-79.197,-175.661,7.687,148.213
C04283=1232.586,400.794,-79.232,-175.660,7.689,148.214
C04284=1232.581,401.042,-79.265,-175.660,7.691,148.214
C04285=1232.578,401.290,-79.300,-175.659,7.694,148.215
C04286=1232.574,401.537,-79.334,-175.658,7.696,148.215
C04287=1232.569,401.785,-79.368,-175.658,7.698,148.215
C04288=1232.565,402.032,-79.401,-175.656,7.700,148.216
C04289=1232.561,402.280,-79.436,-175.656,7.702,148.216
C04290=1232.557,402.528,-79.470,-175.656,7.705,148.217
C04291=1232.553,402.775,-79.505,-175.654,7.708,148.217
C04292=1232.549,403.023,-79.538,-175.654,7.710,148.217
C04293=1232.545,403.271,-79.573,-175.653,7.711,148.218
C04294=1232.541,403.518,-79.606,-175.652,7.714,148.218
C04295=1232.537,403.766,-79.641,-175.652,7.717,148.219
C04296=1232.533,404.014,-79.674,-175.651,7.719,148.219
C04297=1232.528,404.261,-79.709,-175.650,7.721,148.219
C04298=1232.525,404.509,-79.743,-175.649,7.723,148.220
C04299=1232.520,404.756,-79.778,-175.649,7.725,148.220
C04300=1232.516,405.004,-79.811,-175.648,7.728,148.221
C04301=1232.512,405.252,-79.846,-175.647,7.730,148.221
C04302=1232.508,405.499,-79.879,-175.647,7.732,148.221
C04303=1232.504,405.747,-79.914,-175.646,7.734,148.222
C04304=1232.500,405.995,-79.948,-175.645,7.737,148.222
C04305=1232.496,406.242,-79.983,-175.645,7.740,148.223
C04306=1232.492,406.489,-80.016,-175.644,7.741,148.223
C04307=1232.488,406.738,-80.051,-175.644,7.743,148.223
C04308=1232.484,406.985,-80.084,-175.642,7.746,148.224
C04309=1232.479,407.232,-80.119,-175.642,7.748,148.224
C04310=1232.475,407.481,-80.154,-175.642,7.751,148.225
C04311=1232.472,407.728,-80.188,-175.641,7.753,148.225
C04312=1232.467,407.975,-80.222,-175.640,7.755,148.225
C04313=1232.464,408.223,-80.256,-175.639,7.757,148.226
C04314=1232.459,408.471,-80.290,-175.639,7.759,148.226
C04315=1232.455,408.718,-80.324,-175.638,7.762,148.227
C04316=1232.451,408.966,-80.359,-175.637,7.764,148.227
C04317=1232.447,409.214,-80.393,-175.637,7.766,148.227
C04318=1232.443,409.461,-80.427,-175.636,7.768,148.228
C04319=1232.439,409.709,-80.462,-175.635,7.770,148.228
C04320=1232.435,409.956,-80.496,-175.635,7.773,148.229
C04321=1232.431,410.204,-80.531,-175.634,7.775,148.229
C04322=1232.426,410.451,-80.565,-175.633,7.777,148.229
C04323=1232.423,410.699,-80.599,-175.633,7.779,148.230
C04324=1232.419,410.947,-80.634,-175.632,7.781,148.230
C04325=1232.415,411.194,-80.668,-175.631,7.785,148.231
C04326=1232.411,411.442,-80.703,-175.631,7.786,148.231
C04327=1232.406,411.689,-80.737,-175.630,7.788,148.231
C04328=1232.402,411.936,-80.771,-175.630,7.790,148.232
C04329=1232.398,412.185,-80.806,-175.629,7.793,148.232
C04330=1232.394,412.432,-80.840,-175.628,7.796,148.233
C04331=1232.391,412.680,-80.874,-175.628,7.798,148.233
C04332=1232.386,412.927,-80.909,-175.627,7.800,148.233
C04333=1232.381,413.175,-80.943,-175.626,7.801,148.234
C04334=1232.378,413.422,-80.978,-175.626,7.804,148.234
C04335=1232.374,413.670,-81.012,-175.626,7.806,148.234
C04336=1232.370,413.918,-81.046,-175.624,7.809,148.235
C04337=1232.366,414.165,-81.081,-175.624,7.811,148.235
C04338=1232.361,414.412,-81.115,-175.623,7.813,148.236
C04339=1232.357,414.661,-81.150,-175.623,7.815,148.236
C04340=1232.353,414.908,-81.184,-175.622,7.817,148.236
C04341=1232.350,415.156,-81.219,-175.622,7.819,148.237
C04342=1232.345,415.403,-81.253,-175.621,7.821,148.237
C04343=1232.342,415.651,-81.287,-175.620,7.824,148.237
C04344=1232.335,416.013,-81.338,-175.619,7.827,148.238
C04345=1232.330,416.374,-81.388,-175.618,7.830,148.239
C04346=1232.324,416.736,-81.439,-175.618,7.833,148.239
C04347=1232.318,417.097,-81.489,-175.617,7.836,148.240
C04348=1231.896,417.097,-81.521,-175.620,7.846,148.244
C04349=1231.901,416.732,-81.471,-175.621,7.843,148.243
C04350=1231.908,416.368,-81.420,-175.622,7.840,148.242
C04351=1231.913,416.005,-81.369,-175.623,7.837,148.242
C04352=1231.920,415.640,-81.318,-175.624,7.833,148.241
C04353=1231.924,415.392,-81.284,-175.625,7.831,148.241
C04354=1231.928,415.145,-81.250,-175.625,7.829,148.240
C04355=1231.932,414.897,-81.215,-175.625,7.827,148.240
C04356=1231.936,414.650,-81.180,-175.626,7.825,148.240
C04357=1231.939,414.403,-81.145,-175.627,7.823,148.239
C04358=1231.944,414.155,-81.111,-175.627,7.821,148.239
C04359=1231.948,413.908,-81.077,-175.628,7.818,148.238
C04360=1231.951,413.660,-81.042,-175.629,7.816,148.238
C04361=1231.956,413.412,-81.008,-175.629,7.814,148.238
C04362=1231.960,413.164,-80.973,-175.630,7.812,148.237
C04363=1231.964,412.917,-80.939,-175.630,7.810,148.237
C04364=1231.968,412.670,-80.905,-175.631,7.808,148.236
C04365=1231.972,412.422,-80.870,-175.632,7.805,148.236
C04366=1231.976,412.175,-80.836,-175.633,7.803,148.236
C04367=1231.980,411.926,-80.801,-175.633,7.801,148.235
C04368=1231.984,411.679,-80.767,-175.633,7.799,148.235
C04369=1231.988,411.432,-80.733,-175.634,7.797,148.234
C04370=1231.992,411.184,-80.698,-175.635,7.794,148.234
C04371=1231.996,410.937,-80.664,-175.636,7.792,148.234
C04372=1232.000,410.689,-80.629,-175.636,7.790,148.233
C04373=1232.005,410.441,-80.595,-175.637,7.788,148.233
C04374=1232.009,410.194,-80.561,-175.637,7.786,148.233
C04375=1232.013,409.946,-80.526,-175.638,7.783,148.232
C04376=1232.017,409.698,-80.493,-175.639,7.781,148.232
C04377=1232.021,409.450,-80.458,-175.639,7.779,148.231
C04378=1232.025,409.203,-80.424,-175.640,7.777,148.231
C04379=1232.029,408.956,-80.390,-175.640,7.775,148.231
C04380=1232.033,408.707,-80.355,-175.642,7.772,148.230
C04381=1232.037,408.460,-80.321,-175.642,7.770,148.230
C04382=1232.042,408.213,-80.287,-175.642,7.768,148.229
C04383=1232.045,407.965,-80.252,-175.643,7.766,148.229
C04384=1232.049,407.718,-80.218,-175.644,7.763,148.228
C04385=1232.054,407.470,-80.183,-175.645,7.761,148.228
C04386=1232.057,407.222,-80.149,-175.645,7.759,148.228
C04387=1232.062,406.974,-80.115,-175.646,7.757,148.227
C04388=1232.065,406.727,-80.081,-175.647,7.754,148.227
C04389=1232.070,406.479,-80.047,-175.647,7.752,148.227
C04390=1232.074,406.232,-80.013,-175.648,7.750,148.226
C04391=1232.078,405.984,-79.978,-175.648,7.748,148.226
C04392=1232.082,405.737,-79.944,-175.649,7.745,148.225
C04393=1232.086,405.489,-79.910,-175.650,7.743,148.225
C04394=1232.090,405.241,-79.876,-175.651,7.741,148.225
C04395=1232.094,404.994,-79.842,-175.652,7.738,148.224
C04396=1232.099,404.746,-79.807,-175.652,7.736,148.224
C04397=1232.102,404.498,-79.773,-175.653,7.734,148.223
C04398=1232.106,404.251,-79.739,-175.653,7.732,148.223
C04399=1232.111,404.003,-79.705,-175.654,7.729,148.223
C04400=1232.115,403.755,-79.671,-175.655,7.727,148.222
C04401=1232.118,403.508,-79.637,-175.655,7.725,148.222
C04402=1232.123,403.261,-79.602,-175.656,7.722,148.221
C04403=1232.126,403.013,-79.568,-175.657,7.720,148.221
C04404=1232.131,402.765,-79.534,-175.658,7.718,148.221
C04405=1232.135,402.518,-79.500,-175.659,7.715,148.220
C04406=1232.139,402.270,-79.466,-175.659,7.713,148.220
C04407=1232.143,402.022,-79.432,-175.659,7.711,148.219
C04408=1232.148,401.774,-79.398,-175.661,7.708,148.219
C04409=1232.151,401.527,-79.364,-175.661,7.706,148.218
C04410=1232.155,401.279,-79.329,-175.662,7.704,148.218
C04411=1232.160,401.031,-79.296,-175.663,7.701,148.218
C04412=1232.164,400.784,-79.262,-175.663,7.699,148.217
C04413=1232.167,400.536,-79.227,-175.664,7.696,148.217
C04414=1232.172,400.289,-79.193,-175.665,7.694,148.216
C04415=1232.176,400.041,-79.160,-175.666,7.692,148.216
C04416=1232.180,399.794,-79.126,-175.667,7.689,148.216
C04417=1232.184,399.546,-79.091,-175.667,7.687,148.215
C04418=1232.188,399.298,-79.058,-175.668,7.685,148.215
C04419=1232.193,399.051,-79.023,-175.669,7.682,148.214
C04420=1232.196,398.803,-78.989,-175.669,7.680,148.214
C04421=1232.201,398.555,-78.955,-175.671,7.677,148.214
C04422=1232.204,398.308,-78.922,-175.671,7.675,148.213
C04423=1232.208,398.061,-78.888,-175.671,7.673,148.213
C04424=1232.213,397.812,-78.854,-175.673,7.670,148.212
C04425=1232.216,397.565,-78.820,-175.673,7.668,148.212
C04426=1232.221,397.317,-78.786,-175.674,7.666,148.212
C04427=1232.225,397.070,-78.752,-175.675,7.664,148.211
C04428=1232.229,396.821,-78.717,-175.676,7.661,148.211
C04429=1232.233,396.574,-78.684,-175.677,7.659,148.211
C04430=1232.237,396.327,-78.650,-175.677,7.656,148.210
C04431=1232.242,396.079,-78.616,-175.678,7.654,148.210
C04432=1232.245,395.831,-78.582,-175.679,7.652,148.209
C04433=1232.249,395.584,-78.548,-175.680,7.649,148.209
C04434=1232.254,395.336,-78.515,-175.680,7.647,148.209
C04435=1232.258,395.088,-78.481,-175.682,7.644,148.208
C04436=1232.262,394.840,-78.447,-175.682,7.642,148.208
C04437=1232.266,394.593,-78.413,-175.683,7.639,148.207
C04438=1232.270,394.345,-78.380,-175.684,7.637,148.207
C04439=1232.275,394.097,-78.345,-175.685,7.634,148.206
C04440=1232.279,393.850,-78.312,-175.685,7.632,148.206
C04441=1232.283,393.568,-78.273,-175.687,7.629,148.206
C04442=1232.288,393.287,-78.235,-175.688,7.626,148.205
C04443=1232.292,393.006,-78.196,-175.689,7.624,148.205
C04444=1232.297,392.725,-78.158,-175.690,7.621,148.204
C04445=1232.301,392.477,-78.125,-175.690,7.619,148.204
C04446=1232.305,392.229,-78.091,-175.691,7.616,148.203
C04447=1232.309,391.982,-78.057,-175.692,7.614,148.203
C04448=1232.313,391.734,-78.024,-175.693,7.611,148.203
C04449=1232.318,391.486,-77.989,-175.694,7.609,148.202
C04450=1232.321,391.238,-77.956,-175.695,7.606,148.202
C04451=1232.325,390.991,-77.922,-175.696,7.604,148.202
C04452=1232.330,390.743,-77.888,-175.697,7.601,148.201
C04453=1232.334,390.496,-77.854,-175.697,7.599,148.201
C04454=1232.338,390.248,-77.821,-175.698,7.597,148.201
C04455=1232.342,390.000,-77.788,-175.700,7.594,148.200
C04456=1232.346,389.752,-77.753,-175.700,7.591,148.200
C04457=1232.350,389.504,-77.720,-175.701,7.589,148.199
C04458=1232.354,389.257,-77.686,-175.702,7.587,148.199
C04459=1232.358,389.010,-77.653,-175.703,7.584,148.198
C04460=1232.363,388.762,-77.619,-175.703,7.582,148.198
C04461=1232.367,388.515,-77.585,-175.705,7.579,148.198
C04462=1232.370,388.266,-77.552,-175.706,7.576,148.197
C04463=1232.374,388.018,-77.519,-175.706,7.574,148.197
C04464=1232.379,387.771,-77.484,-175.707,7.571,148.197
C04465=1232.383,387.523,-77.451,-175.708,7.569,148.196
C04466=1232.387,387.275,-77.418,-175.709,7.567,148.196
C04467=1232.391,387.028,-77.384,-175.710,7.564,148.195
C04468=1232.395,386.780,-77.350,-175.711,7.562,148.195
C04469=1232.400,386.532,-77.317,-175.712,7.559,148.195
C04470=1232.403,386.285,-77.283,-175.713,7.556,148.194
C04471=1232.408,386.037,-77.250,-175.714,7.554,148.194
C04472=1232.412,385.789,-77.216,-175.715,7.551,148.193
C04473=1232.416,385.542,-77.182,-175.716,7.548,148.193
C04474=1232.420,385.294,-77.149,-175.717,7.546,148.193
C04475=1232.424,385.046,-77.115,-175.718,7.544,148.192
C04476=1232.428,384.798,-77.082,-175.720,7.541,148.192
C04477=1232.432,384.551,-77.048,-175.720,7.539,148.192
C04478=1232.436,384.303,-77.015,-175.721,7.536,148.191
C04479=1232.441,384.055,-76.981,-175.723,7.533,148.191
C04480=1232.445,383.807,-76.948,-175.723,7.531,148.191
C04481=1232.449,383.560,-76.915,-175.724,7.529,148.190
C04482=1232.453,383.313,-76.881,-175.726,7.526,148.190
C04483=1232.457,383.065,-76.848,-175.726,7.524,148.190
C04484=1232.461,382.816,-76.814,-175.727,7.521,148.189
C04485=1232.465,382.569,-76.781,-175.729,7.518,148.189
C04486=1232.470,382.321,-76.748,-175.729,7.516,148.188
C04487=1232.474,382.074,-76.714,-175.730,7.513,148.188
C04488=1232.478,381.826,-76.681,-175.731,7.511,148.188
C04489=1232.482,381.578,-76.647,-175.733,7.508,148.187
C04490=1232.486,381.330,-76.614,-175.734,7.506,148.187
C04491=1232.490,381.083,-76.581,-175.735,7.503,148.187
C04492=1232.494,380.835,-76.548,-175.736,7.500,148.186
C04493=1232.498,380.587,-76.515,-175.737,7.498,148.186
C04494=1232.503,380.339,-76.482,-175.738,7.496,148.185
C04495=1232.506,380.092,-76.448,-175.739,7.493,148.185
C04496=1232.511,379.844,-76.414,-175.741,7.490,148.185
C04497=1232.515,379.596,-76.380,-175.742,7.487,148.184
C04498=1232.519,379.348,-76.347,-175.742,7.485,148.184
C04499=1232.523,379.100,-76.314,-175.744,7.483,148.184
C04500=1232.527,378.853,-76.281,-175.745,7.480,148.183
C04501=1232.531,378.605,-76.248,-175.746,7.477,148.183
C04502=1232.535,378.357,-76.215,-175.747,7.475,148.183
C04503=1232.540,378.109,-76.182,-175.748,7.472,148.182
C04504=1232.544,377.862,-76.148,-175.749,7.470,148.182
C04505=1232.548,377.614,-76.115,-175.750,7.467,148.182
C04506=1232.552,377.366,-76.082,-175.752,7.464,148.181
C04507=1232.556,377.119,-76.049,-175.753,7.462,148.181
C04508=1232.560,376.871,-76.016,-175.754,7.459,148.181
C04509=1232.564,376.623,-75.983,-175.755,7.457,148.180
C04510=1232.569,376.375,-75.949,-175.756,7.454,148.180
C04511=1232.573,376.128,-75.916,-175.758,7.451,148.180
C04512=1232.577,375.880,-75.883,-175.759,7.448,148.179
C04513=1232.581,375.632,-75.850,-175.760,7.446,148.179
C04514=1232.585,375.384,-75.817,-175.761,7.444,148.179
C04515=1232.589,375.137,-75.784,-175.762,7.441,148.178
C04516=1232.593,374.889,-75.751,-175.763,7.438,148.178
C04517=1232.598,374.641,-75.717,-175.765,7.435,148.178
C04518=1232.602,374.394,-75.684,-175.766,7.433,148.177
C04519=1232.606,374.146,-75.651,-175.767,7.431,148.177
C04520=1232.610,373.897,-75.619,-175.768,7.428,148.177
C04521=1232.614,373.650,-75.585,-175.770,7.426,148.176
C04522=1232.619,373.402,-75.552,-175.771,7.423,148.176
C04523=1232.622,373.155,-75.520,-175.772,7.420,148.176
C04524=1232.626,372.907,-75.487,-175.774,7.417,148.175
C04525=1232.630,372.659,-75.453,-175.775,7.414,148.175
C04526=1232.634,372.411,-75.420,-175.776,7.412,148.175
C04527=1232.639,372.163,-75.388,-175.777,7.410,148.175
C04528=1232.643,371.915,-75.355,-175.778,7.407,148.174
C04529=1232.647,371.668,-75.322,-175.779,7.404,148.174
C04530=1232.651,371.420,-75.288,-175.781,7.402,148.174
C04531=1232.655,371.172,-75.255,-175.782,7.399,148.173
C04532=1232.660,370.924,-75.223,-175.783,7.396,148.173
C04533=1232.663,370.676,-75.190,-175.785,7.394,148.173
C04534=1232.667,370.429,-75.157,-175.786,7.391,148.172
C04535=1232.671,370.181,-75.124,-175.788,7.388,148.172
C04536=1232.676,369.933,-75.091,-175.789,7.385,148.172
C04537=1232.680,369.685,-75.058,-175.790,7.383,148.171
C04538=1232.685,369.438,-75.025,-175.792,7.380,148.171
C04539=1232.689,369.190,-74.992,-175.793,7.377,148.171
C04540=1232.693,368.942,-74.960,-175.794,7.375,148.170
C04541=1232.697,368.694,-74.927,-175.795,7.373,148.170
C04542=1232.701,368.447,-74.894,-175.797,7.370,148.170
C04543=1232.705,368.199,-74.861,-175.798,7.367,148.169
C04544=1232.709,367.950,-74.829,-175.799,7.365,148.169
C04545=1232.713,367.671,-74.792,-175.801,7.361,148.169
C04546=1232.719,367.392,-74.754,-175.803,7.359,148.169
C04547=1232.723,367.112,-74.718,-175.804,7.356,148.168
C04548=1232.727,366.833,-74.681,-175.806,7.352,148.168
C04549=1232.732,366.585,-74.649,-175.807,7.350,148.168
C04550=1232.736,366.337,-74.616,-175.809,7.347,148.167
C04551=1232.741,366.090,-74.582,-175.810,7.344,148.167
C04552=1232.744,365.842,-74.551,-175.812,7.342,148.167
C04553=1232.748,365.594,-74.517,-175.813,7.339,148.166
C04554=1232.753,365.346,-74.485,-175.814,7.336,148.166
C04555=1232.757,365.098,-74.452,-175.816,7.334,148.166
C04556=1232.760,364.850,-74.419,-175.817,7.331,148.166
C04557=1232.765,364.603,-74.387,-175.819,7.328,148.165
C04558=1232.770,364.355,-74.354,-175.820,7.326,148.165
C04559=1232.773,364.107,-74.322,-175.821,7.323,148.165
C04560=1232.777,363.859,-74.289,-175.823,7.321,148.165
C04561=1232.782,363.611,-74.257,-175.824,7.318,148.164
C04562=1232.786,363.363,-74.223,-175.826,7.315,148.164
C04563=1232.790,363.115,-74.192,-175.827,7.312,148.164
C04564=1232.795,362.868,-74.159,-175.829,7.310,148.163
C04565=1232.799,362.620,-74.126,-175.830,7.307,148.163
C04566=1232.802,362.372,-74.094,-175.831,7.304,148.163
C04567=1232.807,362.124,-74.061,-175.833,7.302,148.163
C04568=1232.811,361.876,-74.028,-175.835,7.299,148.163
C04569=1232.815,361.628,-73.996,-175.836,7.297,148.162
C04570=1232.819,361.381,-73.964,-175.837,7.294,148.162
C04571=1232.824,361.133,-73.931,-175.839,7.292,148.162
C04572=1232.828,360.885,-73.899,-175.841,7.289,148.162
C04573=1232.832,360.637,-73.866,-175.842,7.286,148.161
C04574=1232.835,360.389,-73.834,-175.844,7.283,148.161
C04575=1232.840,360.141,-73.801,-175.846,7.280,148.161
C04576=1232.845,359.894,-73.769,-175.847,7.277,148.160
C04577=1232.848,359.646,-73.737,-175.848,7.275,148.160
C04578=1232.852,359.398,-73.704,-175.850,7.272,148.160
C04579=1232.857,359.150,-73.672,-175.852,7.270,148.160
C04580=1232.861,358.902,-73.640,-175.853,7.267,148.159
C04581=1232.865,358.655,-73.607,-175.854,7.264,148.159
C04582=1232.869,358.407,-73.575,-175.856,7.262,148.159
C04583=1232.873,358.158,-73.543,-175.858,7.259,148.159
C04584=1232.877,357.911,-73.510,-175.859,7.257,148.159
C04585=1232.882,357.663,-73.478,-175.860,7.254,148.158
C04586=1232.886,357.415,-73.446,-175.863,7.251,148.158
C04587=1232.890,357.167,-73.414,-175.864,7.248,148.158
C04588=1232.894,356.919,-73.381,-175.866,7.246,148.158
C04589=1232.898,356.672,-73.349,-175.867,7.243,148.157
C04590=1232.903,356.423,-73.317,-175.869,7.241,148.157
C04591=1232.907,356.175,-73.285,-175.870,7.238,148.157
C04592=1232.911,355.928,-73.252,-175.872,7.235,148.157
C04593=1232.915,355.680,-73.220,-175.874,7.233,148.156
C04594=1232.920,355.432,-73.188,-175.875,7.230,148.156
C04595=1232.923,355.184,-73.156,-175.877,7.227,148.156
C04596=1232.928,354.935,-73.123,-175.879,7.224,148.156
C04597=1232.932,354.689,-73.091,-175.881,7.222,148.156
C04598=1232.936,354.440,-73.059,-175.882,7.219,148.155
C04599=1232.940,354.192,-73.027,-175.884,7.217,148.155
C04600=1232.945,353.945,-72.995,-175.885,7.214,148.155
C04601=1232.949,353.697,-72.963,-175.887,7.211,148.155
C04602=1232.953,353.448,-72.931,-175.888,7.209,148.155
C04603=1232.957,353.200,-72.899,-175.890,7.205,148.154
C04604=1232.961,352.954,-72.867,-175.892,7.203,148.154
C04605=1232.965,352.705,-72.834,-175.894,7.200,148.154
C04606=1232.969,352.457,-72.802,-175.895,7.198,148.154
C04607=1232.974,352.210,-72.770,-175.897,7.195,148.154
C04608=1232.978,351.961,-72.738,-175.898,7.193,148.153
C04609=1232.982,351.713,-72.706,-175.900,7.190,148.153
C04610=1232.986,351.466,-72.674,-175.902,7.188,148.153
C04611=1232.990,351.218,-72.643,-175.904,7.184,148.153
C04612=1232.995,350.969,-72.610,-175.905,7.182,148.153
C04613=1232.999,350.722,-72.579,-175.907,7.179,148.152
C04614=1233.003,350.474,-72.546,-175.909,7.177,148.152
C04615=1233.007,350.226,-72.514,-175.910,7.174,148.152
C04616=1233.011,349.978,-72.483,-175.912,7.172,148.152
C04617=1233.016,349.730,-72.450,-175.914,7.168,148.152
C04618=1233.019,349.482,-72.419,-175.916,7.166,148.151
C04619=1233.024,349.235,-72.387,-175.917,7.163,148.151
C04620=1233.028,348.986,-72.355,-175.919,7.161,148.151
C04621=1233.032,348.738,-72.323,-175.921,7.158,148.151
C04622=1233.036,348.491,-72.291,-175.922,7.156,148.151
C04623=1233.041,348.243,-72.259,-175.925,7.152,148.151
C04624=1233.045,347.995,-72.227,-175.926,7.150,148.150
C04625=1233.049,347.747,-72.196,-175.928,7.147,148.150
C04626=1233.053,347.498,-72.164,-175.930,7.145,148.150
C04627=1233.058,347.251,-72.132,-175.931,7.142,148.150
C04628=1233.061,347.003,-72.101,-175.933,7.140,148.150
C04629=1233.065,346.755,-72.069,-175.935,7.136,148.150
C04630=1233.070,346.507,-72.037,-175.937,7.134,148.149
C04631=1233.074,346.259,-72.005,-175.938,7.131,148.149
C04632=1233.078,346.011,-71.974,-175.940,7.129,148.149
C04633=1233.083,345.763,-71.942,-175.942,7.127,148.149
C04634=1233.087,345.515,-71.910,-175.944,7.124,148.149
C04635=1233.091,345.267,-71.878,-175.946,7.121,148.149
C04636=1233.095,345.019,-71.846,-175.947,7.118,148.148
C04637=1233.100,344.771,-71.815,-175.949,7.116,148.148
C04638=1233.104,344.523,-71.783,-175.951,7.113,148.148
C04639=1233.108,344.276,-71.752,-175.953,7.111,148.148
C04640=1233.112,344.028,-71.720,-175.955,7.107,148.148
C04641=1233.116,343.780,-71.689,-175.957,7.105,148.148
C04642=1233.121,343.531,-71.657,-175.958,7.102,148.147
C04643=1233.125,343.284,-71.625,-175.960,7.100,148.148
C04644=1233.129,343.035,-71.594,-175.962,7.098,148.147
C04645=1233.133,342.787,-71.562,-175.964,7.094,148.147
C04646=1233.137,342.540,-71.531,-175.966,7.092,148.147
C04647=1233.141,342.291,-71.500,-175.968,7.089,148.147
C04648=1233.146,342.044,-71.468,-175.969,7.087,148.147
C04649=1233.151,341.766,-71.432,-175.972,7.084,148.147
C04650=1233.156,341.489,-71.397,-175.973,7.081,148.146
C04651=1233.160,341.211,-71.362,-175.976,7.078,148.146
C04652=1233.164,340.934,-71.326,-175.977,7.075,148.146
C04653=1233.169,340.686,-71.295,-175.980,7.072,148.146
C04654=1233.173,340.438,-71.264,-175.982,7.070,148.146
C04655=1233.177,340.190,-71.233,-175.983,7.067,148.146
C04656=1233.181,339.942,-71.201,-175.985,7.065,148.146
C04657=1233.186,339.694,-71.170,-175.988,7.062,148.146
C04658=1233.190,339.445,-71.138,-175.989,7.059,148.145
C04659=1233.194,339.198,-71.106,-175.991,7.057,148.145
C04660=1233.198,338.949,-71.075,-175.993,7.054,148.145
C04661=1233.203,338.702,-71.044,-175.995,7.052,148.145
C04662=1233.207,338.453,-71.013,-175.997,7.048,148.145
C04663=1233.211,338.206,-70.981,-175.999,7.046,148.145
C04664=1233.216,337.958,-70.950,-176.000,7.044,148.145
C04665=1233.219,337.710,-70.918,-176.002,7.041,148.145
C04666=1233.224,337.462,-70.888,-176.004,7.039,148.145
C04667=1233.228,337.213,-70.857,-176.006,7.036,148.144
C04668=1233.232,336.966,-70.825,-176.008,7.033,148.144
C04669=1233.236,336.717,-70.794,-176.010,7.031,148.144
C04670=1233.241,336.470,-70.762,-176.012,7.028,148.144
C04671=1233.245,336.221,-70.731,-176.014,7.025,148.144
C04672=1233.249,335.974,-70.700,-176.016,7.023,148.144
C04673=1233.254,335.726,-70.669,-176.018,7.020,148.144
C04674=1233.258,335.477,-70.638,-176.020,7.018,148.144
C04675=1233.262,335.230,-70.606,-176.021,7.015,148.143
C04676=1233.266,334.981,-70.575,-176.024,7.012,148.143
C04677=1233.270,334.734,-70.545,-176.025,7.010,148.143
C04678=1233.274,334.485,-70.513,-176.028,7.008,148.143
C04679=1233.279,334.238,-70.482,-176.029,7.005,148.143
C04680=1233.283,333.990,-70.451,-176.032,7.002,148.143
C04681=1233.287,333.742,-70.419,-176.033,6.999,148.143
C04682=1233.291,333.494,-70.389,-176.036,6.997,148.143
C04683=1233.295,333.245,-70.358,-176.037,6.995,148.143
C04684=1233.300,332.997,-70.327,-176.040,6.992,148.143
C04685=1233.304,332.750,-70.296,-176.041,6.989,148.143
C04686=1233.308,332.501,-70.265,-176.044,6.987,148.143
C04687=1233.313,332.253,-70.234,-176.045,6.984,148.142
C04688=1233.317,332.005,-70.203,-176.047,6.982,148.143
C04689=1233.321,331.757,-70.171,-176.049,6.979,148.142
C04690=1233.325,331.509,-70.141,-176.052,6.976,148.142
C04691=1233.329,331.262,-70.110,-176.053,6.974,148.142
C04692=1233.333,331.013,-70.079,-176.055,6.972,148.142
C04693=1233.338,330.765,-70.049,-176.057,6.968,148.142
C04694=1233.342,330.518,-70.017,-176.059,6.966,148.142
C04695=1233.346,330.269,-69.986,-176.061,6.964,148.142
C04696=1233.351,330.021,-69.955,-176.063,6.961,148.142
C04697=1233.356,329.773,-69.924,-176.066,6.958,148.142
C04698=1233.359,329.525,-69.894,-176.067,6.956,148.142
C04699=1233.363,329.277,-69.863,-176.070,6.953,148.142
C04700=1233.368,329.029,-69.832,-176.071,6.951,148.142
C04701=1233.372,328.780,-69.801,-176.074,6.948,148.142
C04702=1233.376,328.533,-69.771,-176.075,6.945,148.141
C04703=1233.380,328.285,-69.740,-176.078,6.943,148.141
C04704=1233.384,328.037,-69.708,-176.080,6.941,148.141
C04705=1233.389,327.789,-69.678,-176.081,6.938,148.141
C04706=1233.393,327.541,-69.647,-176.084,6.935,148.141
C04707=1233.397,327.292,-69.616,-176.086,6.933,148.141
C04708=1233.401,327.044,-69.586,-176.088,6.930,148.141
C04709=1233.406,326.796,-69.555,-176.090,6.928,148.141
C04710=1233.410,326.549,-69.525,-176.092,6.925,148.141
C04711=1233.414,326.300,-69.494,-176.094,6.923,148.141
C04712=1233.418,326.052,-69.463,-176.096,6.920,148.141
C04713=1233.423,325.804,-69.432,-176.098,6.918,148.141
C04714=1233.427,325.557,-69.402,-176.100,6.915,148.141
C04715=1233.431,325.307,-69.371,-176.102,6.913,148.141
C04716=1233.436,325.059,-69.341,-176.104,6.910,148.141
C04717=1233.440,324.812,-69.310,-176.106,6.908,148.141
C04718=1233.444,324.563,-69.279,-176.109,6.905,148.141
C04719=1233.448,324.315,-69.249,-176.111,6.903,148.141
C04720=1233.452,324.067,-69.218,-176.112,6.900,148.141
C04721=1233.457,323.819,-69.188,-176.115,6.898,148.141
C04722=1233.461,323.572,-69.157,-176.117,6.895,148.141
C04723=1233.465,323.323,-69.126,-176.119,6.892,148.140
C04724=1233.470,323.075,-69.096,-176.121,6.890,148.141
C04725=1233.474,322.827,-69.066,-176.123,6.888,148.141
C04726=1233.478,322.579,-69.035,-176.126,6.885,148.141
C04727=1233.482,322.330,-69.004,-176.127,6.882,148.140
C04728=1233.486,322.083,-68.974,-176.129,6.880,148.140
C04729=1233.491,321.834,-68.944,-176.131,6.878,148.140
C04730=1233.495,321.586,-68.914,-176.134,6.875,148.140
C04731=1233.499,321.338,-68.883,-176.136,6.872,148.140
C04732=1233.503,321.090,-68.852,-176.138,6.870,148.140
C04733=1233.508,320.842,-68.822,-176.140,6.868,148.140
C04734=1233.512,320.594,-68.792,-176.142,6.865,148.140
C04735=1233.516,320.346,-68.762,-176.144,6.862,148.140
C04736=1233.521,320.098,-68.731,-176.146,6.860,148.140
C04737=1233.525,319.850,-68.701,-176.148,6.858,148.140
C04738=1233.529,319.601,-68.670,-176.150,6.855,148.140
C04739=1233.533,319.353,-68.640,-176.153,6.852,148.140
C04740=1233.538,319.105,-68.610,-176.155,6.850,148.140
C04741=1233.542,318.857,-68.580,-176.157,6.847,148.140
C04742=1233.546,318.609,-68.549,-176.159,6.845,148.140
C04743=1233.550,318.361,-68.520,-176.162,6.842,148.140
C04744=1233.555,318.113,-68.489,-176.164,6.840,148.140
C04745=1233.559,317.864,-68.459,-176.166,6.838,148.140
C04746=1233.563,317.616,-68.428,-176.167,6.835,148.140
C04747=1233.567,317.368,-68.398,-176.170,6.832,148.140
C04748=1233.572,317.120,-68.368,-176.172,6.830,148.140
C04749=1233.576,316.872,-68.338,-176.174,6.828,148.140
C04750=1233.581,316.624,-68.308,-176.176,6.825,148.140
C04751=1233.585,316.376,-68.278,-176.179,6.822,148.140
C04752=1233.590,316.127,-68.248,-176.181,6.820,148.140
C04753=1233.594,315.852,-68.214,-176.183,6.818,148.140
C04754=1233.598,315.576,-68.181,-176.186,6.815,148.140
C04755=1233.603,315.301,-68.147,-176.188,6.811,148.140
C04756=1233.608,315.025,-68.114,-176.190,6.809,148.140
C04757=1233.612,314.777,-68.083,-176.192,6.807,148.140
C04758=1233.616,314.528,-68.054,-176.195,6.804,148.140
C04759=1233.620,314.281,-68.024,-176.197,6.802,148.140
C04760=1233.625,314.032,-67.994,-176.199,6.799,148.140
C04761=1233.629,313.785,-67.963,-176.201,6.797,148.140
C04762=1233.634,313.536,-67.933,-176.204,6.794,148.140
C04763=1233.638,313.288,-67.904,-176.206,6.792,148.140
C04764=1233.642,313.040,-67.874,-176.208,6.790,148.140
C04765=1233.647,312.791,-67.844,-176.210,6.788,148.141
C04766=1233.651,312.543,-67.814,-176.213,6.784,148.141
C04767=1233.655,312.296,-67.784,-176.215,6.782,148.141
C04768=1233.660,312.047,-67.754,-176.217,6.780,148.141
C04769=1233.664,311.799,-67.724,-176.219,6.778,148.141
C04770=1233.668,311.551,-67.694,-176.221,6.776,148.141
C04771=1233.672,311.302,-67.665,-176.224,6.772,148.141
C04772=1233.677,311.054,-67.635,-176.226,6.770,148.141
C04773=1233.680,310.806,-67.604,-176.228,6.768,148.141
C04774=1233.685,310.558,-67.575,-176.230,6.766,148.141
C04775=1233.690,310.309,-67.545,-176.232,6.762,148.141
C04776=1233.693,310.061,-67.515,-176.234,6.760,148.141
C04777=1233.698,309.813,-67.485,-176.236,6.758,148.141
C04778=1233.702,309.566,-67.456,-176.239,6.756,148.141
C04779=1233.707,309.317,-67.426,-176.242,6.753,148.141
C04780=1233.712,309.069,-67.397,-176.244,6.751,148.141
C04781=1233.715,308.821,-67.367,-176.246,6.749,148.141
C04782=1233.720,308.573,-67.337,-176.248,6.746,148.141
C04783=1233.724,308.325,-67.308,-176.250,6.744,148.141
C04784=1233.729,308.076,-67.278,-176.253,6.741,148.141
C04785=1233.733,307.828,-67.248,-176.255,6.739,148.141
C04786=1233.737,307.580,-67.218,-176.257,6.737,148.141
C04787=1233.741,307.332,-67.189,-176.259,6.734,148.141
C04788=1233.745,307.084,-67.159,-176.262,6.731,148.141
C04789=1233.749,306.835,-67.130,-176.264,6.729,148.141
C04790=1233.754,306.587,-67.100,-176.266,6.727,148.141
C04791=1233.758,306.338,-67.070,-176.268,6.725,148.142
C04792=1233.763,306.090,-67.041,-176.270,6.722,148.142
C04793=1233.767,305.842,-67.011,-176.273,6.719,148.142
C04794=1233.771,305.594,-66.982,-176.275,6.717,148.142
C04795=1233.775,305.345,-66.952,-176.277,6.715,148.142
C04796=1233.780,305.098,-66.923,-176.279,6.713,148.142
C04797=1233.785,304.849,-66.893,-176.282,6.710,148.142
C04798=1233.789,304.601,-66.864,-176.284,6.708,148.142
C04799=1233.793,304.353,-66.834,-176.286,6.705,148.142
C04800=1233.797,304.104,-66.805,-176.288,6.703,148.142
C04801=1233.802,303.856,-66.775,-176.290,6.701,148.142
C04802=1233.806,303.608,-66.746,-176.293,6.698,148.142
C04803=1233.810,303.360,-66.716,-176.295,6.696,148.142
C04804=1233.814,303.111,-66.687,-176.297,6.693,148.142
C04805=1233.819,302.864,-66.658,-176.299,6.691,148.142
C04806=1233.823,302.615,-66.628,-176.302,6.689,148.143
C04807=1233.827,302.367,-66.599,-176.305,6.686,148.143
C04808=1233.831,302.119,-66.570,-176.307,6.684,148.143
C04809=1233.836,301.871,-66.540,-176.309,6.682,148.143
C04810=1233.840,301.622,-66.511,-176.311,6.680,148.143
C04811=1233.844,301.374,-66.481,-176.313,6.677,148.143
C04812=1233.849,301.126,-66.453,-176.316,6.674,148.143
C04813=1233.853,300.878,-66.423,-176.318,6.672,148.143
C04814=1233.857,300.629,-66.394,-176.320,6.670,148.143
C04815=1233.862,300.381,-66.364,-176.323,6.668,148.143
C04816=1233.866,300.133,-66.335,-176.325,6.665,148.143
C04817=1233.870,299.885,-66.306,-176.327,6.663,148.143
C04818=1233.875,299.636,-66.277,-176.330,6.661,148.144
C04819=1233.879,299.388,-66.248,-176.332,6.658,148.144
C04820=1233.883,299.140,-66.218,-176.334,6.656,148.144
C04821=1233.888,298.892,-66.189,-176.336,6.654,148.144
C04822=1233.892,298.643,-66.160,-176.339,6.651,148.144
C04823=1233.897,298.395,-66.131,-176.341,6.649,148.144
C04824=1233.901,298.147,-66.102,-176.343,6.647,148.144
C04825=1233.905,297.899,-66.072,-176.346,6.645,148.144
C04826=1233.909,297.650,-66.044,-176.348,6.642,148.144
C04827=1233.913,297.402,-66.014,-176.350,6.639,148.144
C04828=1233.918,297.154,-65.985,-176.353,6.637,148.144
C04829=1233.922,296.905,-65.957,-176.355,6.635,148.145
C04830=1233.927,296.657,-65.927,-176.357,6.633,148.145
C04831=1233.931,296.409,-65.898,-176.359,6.631,148.145
C04832=1233.936,296.161,-65.869,-176.362,6.628,148.145
C04833=1233.939,295.913,-65.841,-176.364,6.626,148.145
C04834=1233.944,295.664,-65.812,-176.367,6.624,148.145
C04835=1233.948,295.416,-65.782,-176.369,6.621,148.145
C04836=1233.953,295.168,-65.753,-176.371,6.619,148.145
C04837=1233.957,294.919,-65.725,-176.374,6.616,148.145
C04838=1233.961,294.671,-65.695,-176.376,6.614,148.145
C04839=1233.965,294.422,-65.667,-176.378,6.612,148.145
C04840=1233.970,294.175,-65.638,-176.381,6.610,148.146
C04841=1233.974,293.926,-65.609,-176.383,6.608,148.146
C04842=1233.979,293.677,-65.580,-176.385,6.606,148.146
C04843=1233.983,293.430,-65.551,-176.388,6.603,148.146
C04844=1233.987,293.181,-65.522,-176.390,6.601,148.146
C04845=1233.991,292.933,-65.493,-176.392,6.598,148.146
C04846=1233.996,292.685,-65.465,-176.394,6.596,148.146
C04847=1234.000,292.436,-65.436,-176.397,6.594,148.147
C04848=1234.004,292.188,-65.407,-176.399,6.592,148.147
C04849=1234.009,291.939,-65.378,-176.402,6.589,148.147
C04850=1234.014,291.692,-65.349,-176.404,6.587,148.147
C04851=1234.017,291.443,-65.321,-176.406,6.585,148.147
C04852=1234.022,291.195,-65.292,-176.408,6.583,148.147
C04853=1234.027,290.947,-65.263,-176.411,6.581,148.147
C04854=1234.030,290.698,-65.235,-176.413,6.578,148.147
C04855=1234.035,290.450,-65.206,-176.416,6.575,148.147
C04856=1234.040,290.202,-65.177,-176.418,6.573,148.148
C04857=1234.044,289.927,-65.146,-176.421,6.571,148.148
C04858=1234.049,289.653,-65.113,-176.424,6.568,148.148
C04859=1234.054,289.380,-65.083,-176.426,6.566,148.148
C04860=1234.058,289.106,-65.051,-176.429,6.563,148.148
C04861=1234.063,288.857,-65.022,-176.431,6.561,148.148
C04862=1234.068,288.609,-64.993,-176.433,6.559,148.148
C04863=1234.071,288.361,-64.965,-176.436,6.557,148.149
C04864=1234.076,288.112,-64.936,-176.438,6.555,148.149
C04865=1234.080,287.864,-64.908,-176.440,6.553,148.149
C04866=1234.084,287.616,-64.879,-176.443,6.550,148.149
C04867=1234.090,287.368,-64.851,-176.445,6.548,148.149
C04868=1234.093,287.119,-64.822,-176.448,6.546,148.149
C04869=1234.098,286.870,-64.794,-176.450,6.544,148.149
C04870=1234.102,286.622,-64.766,-176.452,6.541,148.149
C04871=1234.106,286.374,-64.736,-176.455,6.539,148.150
C04872=1234.111,286.126,-64.709,-176.457,6.536,148.150
C04873=1234.115,285.877,-64.680,-176.460,6.534,148.150
C04874=1234.120,285.628,-64.651,-176.462,6.532,148.150
C04875=1234.124,285.380,-64.623,-176.464,6.530,148.150
C04876=1234.129,285.131,-64.595,-176.467,6.528,148.150
C04877=1234.133,284.884,-64.566,-176.469,6.526,148.151
C04878=1234.137,284.635,-64.537,-176.471,6.524,148.151
C04879=1234.141,284.387,-64.510,-176.473,6.522,148.151
C04880=1234.146,284.139,-64.481,-176.477,6.519,148.151
C04881=1234.150,283.891,-64.453,-176.479,6.517,148.151
C04882=1234.155,283.642,-64.424,-176.481,6.515,148.151
C04883=1234.159,283.394,-64.397,-176.483,6.513,148.152
C04884=1234.164,283.145,-64.368,-176.485,6.510,148.152
C04885=1234.168,282.897,-64.340,-176.488,6.509,148.152
C04886=1234.172,282.648,-64.311,-176.490,6.506,148.152
C04887=1234.177,282.400,-64.284,-176.493,6.504,148.152
C04888=1234.180,282.152,-64.256,-176.495,6.501,148.152
C04889=1234.186,281.904,-64.227,-176.498,6.499,148.153
C04890=1234.189,281.655,-64.199,-176.500,6.497,148.153
C04891=1234.194,281.407,-64.171,-176.502,6.495,148.153
C04892=1234.198,281.158,-64.142,-176.505,6.493,148.153
C04893=1234.203,280.910,-64.115,-176.507,6.491,148.153
C04894=1234.207,280.662,-64.086,-176.509,6.489,148.153
C04895=1234.211,280.414,-64.058,-176.512,6.487,148.153
C04896=1234.216,280.165,-64.029,-176.515,6.484,148.154
C04897=1234.220,279.917,-64.002,-176.517,6.482,148.154
C04898=1234.224,279.668,-63.974,-176.519,6.480,148.154
C04899=1234.229,279.420,-63.945,-176.522,6.478,148.154
C04900=1234.233,279.171,-63.918,-176.524,6.476,148.154
C04901=1234.237,278.923,-63.890,-176.526,6.474,148.154
C04902=1234.242,278.674,-63.861,-176.529,6.472,148.155
C04903=1234.246,278.426,-63.833,-176.531,6.469,148.155
C04904=1234.250,278.178,-63.805,-176.534,6.468,148.155
C04905=1234.255,277.930,-63.777,-176.536,6.464,148.155
C04906=1234.259,277.682,-63.749,-176.539,6.463,148.155
C04907=1234.264,277.432,-63.722,-176.541,6.460,148.155
C04908=1234.269,277.184,-63.693,-176.543,6.458,148.156
C04909=1234.272,276.936,-63.665,-176.546,6.456,148.156
C04910=1234.277,276.688,-63.637,-176.548,6.454,148.156
C04911=1234.281,276.439,-63.610,-176.550,6.452,148.156
C04912=1234.286,276.190,-63.582,-176.553,6.450,148.156
C04913=1234.290,275.943,-63.554,-176.555,6.448,148.157
C04914=1234.294,275.694,-63.526,-176.558,6.446,148.157
C04915=1234.299,275.446,-63.499,-176.560,6.444,148.157
C04916=1234.304,275.197,-63.470,-176.563,6.441,148.157
C04917=1234.307,274.949,-63.442,-176.565,6.439,148.157
C04918=1234.312,274.700,-63.415,-176.568,6.437,148.157
C04919=1234.316,274.452,-63.387,-176.570,6.435,148.158
C04920=1234.321,274.203,-63.359,-176.572,6.433,148.158
C04921=1234.326,273.955,-63.331,-176.575,6.431,148.158
C04922=1234.329,273.706,-63.303,-176.577,6.429,148.158
C04923=1234.334,273.459,-63.276,-176.580,6.427,148.159
C04924=1234.338,273.210,-63.249,-176.582,6.425,148.159
C04925=1234.343,272.961,-63.220,-176.584,6.423,148.159
C04926=1234.348,272.713,-63.193,-176.587,6.421,148.159
C04927=1234.352,272.465,-63.165,-176.589,6.419,148.159
C04928=1234.356,272.216,-63.138,-176.592,6.417,148.160
C04929=1234.360,271.968,-63.110,-176.594,6.414,148.160
C04930=1234.365,271.720,-63.082,-176.597,6.412,148.160
C04931=1234.369,271.471,-63.055,-176.599,6.410,148.160
C04932=1234.374,271.222,-63.026,-176.602,6.408,148.160
C04933=1234.378,270.974,-62.999,-176.604,6.406,148.160
C04934=1234.382,270.725,-62.971,-176.606,6.404,148.161
C04935=1234.387,270.477,-62.944,-176.609,6.402,148.161
C04936=1234.391,270.229,-62.916,-176.611,6.400,148.161
C04937=1234.395,269.980,-62.889,-176.614,6.398,148.161
C04938=1234.400,269.731,-62.862,-176.616,6.396,148.162
C04939=1234.404,269.483,-62.834,-176.618,6.393,148.162
C04940=1234.409,269.235,-62.807,-176.621,6.391,148.162
C04941=1234.413,268.986,-62.779,-176.623,6.390,148.162
C04942=1234.417,268.738,-62.752,-176.626,6.387,148.162
C04943=1234.422,268.490,-62.724,-176.628,6.385,148.163
C04944=1234.426,268.242,-62.697,-176.631,6.384,148.163
C04945=1234.430,267.992,-62.669,-176.633,6.381,148.163
C04946=1234.435,267.744,-62.642,-176.636,6.379,148.163
C04947=1234.439,267.496,-62.614,-176.638,6.376,148.163
C04948=1234.444,267.247,-62.587,-176.641,6.374,148.164
C04949=1234.448,266.999,-62.559,-176.643,6.373,148.164
C04950=1234.452,266.750,-62.532,-176.645,6.370,148.164
C04951=1234.457,266.502,-62.505,-176.648,6.368,148.164
C04952=1234.461,266.254,-62.477,-176.651,6.367,148.165
C04953=1234.465,266.005,-62.450,-176.653,6.364,148.165
C04954=1234.470,265.756,-62.423,-176.655,6.362,148.165
C04955=1234.475,265.508,-62.396,-176.658,6.361,148.165
C04956=1234.479,265.260,-62.368,-176.660,6.358,148.165
C04957=1234.484,265.011,-62.341,-176.663,6.356,148.166
C04958=1234.488,264.762,-62.314,-176.665,6.355,148.166
C04959=1234.493,264.514,-62.286,-176.667,6.352,148.166
C04960=1234.497,264.266,-62.259,-176.670,6.350,148.166
C04961=1234.502,263.993,-62.230,-176.673,6.349,148.167
C04962=1234.507,263.720,-62.199,-176.676,6.346,148.167
C04963=1234.511,263.448,-62.170,-176.678,6.344,148.167
C04964=1234.517,263.175,-62.139,-176.680,6.342,148.167
C04965=1234.521,262.927,-62.113,-176.683,6.340,148.167
C04966=1234.525,262.678,-62.085,-176.686,6.338,148.168
C04967=1234.529,262.430,-62.058,-176.688,6.336,148.168
C04968=1234.534,262.181,-62.031,-176.690,6.334,148.168
C04969=1234.539,261.933,-62.004,-176.693,6.332,148.168
C04970=1234.543,261.685,-61.977,-176.695,6.330,148.169
C04971=1234.548,261.436,-61.949,-176.698,6.328,148.169
C04972=1234.552,261.188,-61.923,-176.700,6.326,148.169
C04973=1234.556,260.939,-61.896,-176.702,6.324,148.169
C04974=1234.560,260.690,-61.869,-176.705,6.322,148.169
C04975=1234.565,260.442,-61.841,-176.708,6.320,148.170
C04976=1234.570,260.193,-61.814,-176.710,6.318,148.170
C04977=1234.574,259.945,-61.788,-176.712,6.316,148.170
C04978=1234.578,259.697,-61.761,-176.715,6.314,148.170
C04979=1234.583,259.448,-61.734,-176.717,6.312,148.171
C04980=1234.588,259.200,-61.707,-176.720,6.310,148.171
C04981=1234.592,258.950,-61.679,-176.722,6.308,148.171
C04982=1234.596,258.702,-61.653,-176.725,6.306,148.171
C04983=1234.600,258.454,-61.626,-176.727,6.304,148.172
C04984=1234.605,258.205,-61.599,-176.730,6.302,148.172
C04985=1234.609,257.957,-61.572,-176.732,6.300,148.172
C04986=1234.613,257.709,-61.545,-176.735,6.298,148.172
C04987=1234.618,257.460,-61.518,-176.737,6.296,148.173
C04988=1234.623,257.211,-61.492,-176.739,6.294,148.173
C04989=1234.627,256.963,-61.465,-176.742,6.292,148.173
C04990=1234.632,256.714,-61.438,-176.745,6.290,148.173
C04991=1234.636,256.466,-61.411,-176.747,6.288,148.174
C04992=1234.640,256.218,-61.385,-176.749,6.286,148.174
C04993=1234.645,255.969,-61.358,-176.752,6.284,148.174
C04994=1234.649,255.721,-61.331,-176.755,6.282,148.174
C04995=1234.654,255.472,-61.305,-176.757,6.280,148.175
C04996=1234.658,255.223,-61.278,-176.759,6.278,148.175
C04997=1234.663,254.975,-61.251,-176.762,6.276,148.175
C04998=1234.666,254.726,-61.224,-176.765,6.274,148.175
C04999=1234.671,254.477,-61.197,-176.767,6.272,148.176
C05000=1234.676,254.228,-61.170,-176.769,6.270,148.176
C05001=1234.680,253.980,-61.144,-176.772,6.268,148.176
C05002=1234.685,253.732,-61.117,-176.774,6.266,148.176
C05003=1234.689,253.483,-61.090,-176.777,6.265,148.177
C05004=1234.693,253.234,-61.064,-176.779,6.262,148.177
C05005=1234.698,252.986,-61.037,-176.782,6.260,148.177
C05006=1234.702,252.738,-61.011,-176.784,6.259,148.177
C05007=1234.707,252.489,-60.984,-176.787,6.257,148.178
C05008=1234.711,252.240,-60.958,-176.790,6.255,148.178
C05009=1234.716,251.992,-60.931,-176.792,6.253,148.178
C05010=1234.721,251.743,-60.905,-176.794,6.251,148.178
C05011=1234.725,251.495,-60.878,-176.797,6.249,148.179
C05012=1234.730,251.247,-60.851,-176.800,6.247,148.179
C05013=1234.734,250.998,-60.825,-176.802,6.245,148.179
C05014=1234.739,250.749,-60.798,-176.804,6.244,148.179
C05015=1234.742,250.501,-60.772,-176.806,6.242,148.180
C05016=1234.747,250.252,-60.746,-176.809,6.240,148.180
C05017=1234.751,250.004,-60.719,-176.812,6.238,148.180
C05018=1234.756,249.755,-60.693,-176.814,6.236,148.181
C05019=1234.760,249.507,-60.666,-176.816,6.234,148.181
C05020=1234.765,249.258,-60.640,-176.819,6.232,148.181
C05021=1234.769,249.009,-60.614,-176.821,6.230,148.181
C05022=1234.774,248.761,-60.586,-176.824,6.228,148.182
C05023=1234.778,248.512,-60.561,-176.827,6.226,148.182
C05024=1234.783,248.264,-60.534,-176.829,6.224,148.182
C05025=1234.787,248.015,-60.508,-176.831,6.222,148.182
C05026=1234.791,247.767,-60.482,-176.834,6.220,148.183
C05027=1234.796,247.518,-60.455,-176.837,6.218,148.183
C05028=1234.801,247.269,-60.430,-176.839,6.217,148.183
C05029=1234.805,247.021,-60.403,-176.842,6.215,148.184
C05030=1234.809,246.772,-60.377,-176.843,6.213,148.184
C05031=1234.814,246.524,-60.350,-176.846,6.211,148.184
C05032=1234.818,246.275,-60.324,-176.849,6.210,148.184
C05033=1234.822,246.027,-60.298,-176.851,6.208,148.185
C05034=1234.828,245.778,-60.272,-176.854,6.206,148.185
C05035=1234.832,245.529,-60.246,-176.856,6.204,148.185
C05036=1234.836,245.281,-60.219,-176.859,6.202,148.186
C05037=1234.841,245.032,-60.193,-176.861,6.200,148.186
C05038=1234.845,244.784,-60.167,-176.864,6.198,148.186
C05039=1234.850,244.535,-60.140,-176.866,6.196,148.186
C05040=1234.854,244.286,-60.115,-176.869,6.194,148.187
C05041=1234.859,244.038,-60.088,-176.872,6.192,148.187
C05042=1234.864,243.789,-60.062,-176.874,6.190,148.187
C05043=1234.868,243.541,-60.036,-176.876,6.189,148.188
C05044=1234.872,243.292,-60.011,-176.878,6.187,148.188
C05045=1234.876,243.044,-59.984,-176.881,6.185,148.188
C05046=1234.881,242.794,-59.958,-176.884,6.183,148.188
C05047=1234.886,242.546,-59.932,-176.886,6.181,148.189
C05048=1234.890,242.298,-59.906,-176.889,6.180,148.189
C05049=1234.895,242.049,-59.880,-176.891,6.178,148.189
C05050=1234.899,241.800,-59.854,-176.894,6.176,148.190
C05051=1234.903,241.551,-59.828,-176.897,6.174,148.190
C05052=1234.908,241.303,-59.803,-176.899,6.172,148.190
C05053=1234.913,241.055,-59.776,-176.901,6.171,148.190
C05054=1234.917,240.806,-59.750,-176.903,6.169,148.191
C05055=1234.921,240.557,-59.724,-176.906,6.167,148.191
C05056=1234.926,240.309,-59.699,-176.909,6.165,148.191
C05057=1234.931,240.060,-59.672,-176.911,6.163,148.192
C05058=1234.935,239.811,-59.647,-176.914,6.161,148.192
C05059=1234.939,239.563,-59.620,-176.917,6.159,148.192
C05060=1234.943,239.314,-59.594,-176.919,6.157,148.193
C05061=1234.948,239.066,-59.569,-176.921,6.155,148.193
C05062=1234.953,238.817,-59.543,-176.923,6.154,148.193
C05063=1234.957,238.568,-59.517,-176.926,6.152,148.193
C05064=1234.962,238.320,-59.492,-176.929,6.150,148.194
C05065=1234.967,238.048,-59.463,-176.931,6.149,148.194
C05066=1234.971,237.777,-59.435,-176.934,6.146,148.194
C05067=1234.976,237.506,-59.407,-176.937,6.144,148.194
C05068=1234.981,237.234,-59.379,-176.940,6.142,148.195
C05069=1234.986,236.986,-59.354,-176.942,6.140,148.195
C05070=1234.990,236.737,-59.328,-176.945,6.138,148.195
C05071=1234.995,236.488,-59.302,-176.947,6.137,148.196
C05072=1234.999,236.239,-59.276,-176.949,6.135,148.196
C05073=1235.004,235.991,-59.250,-176.952,6.133,148.196
C05074=1235.008,235.742,-59.225,-176.955,6.132,148.197
C05075=1235.013,235.493,-59.199,-176.957,6.130,148.197
C05076=1235.017,235.245,-59.174,-176.960,6.128,148.197
C05077=1235.022,234.996,-59.148,-176.963,6.126,148.198
C05078=1235.026,234.748,-59.122,-176.965,6.124,148.198
C05079=1235.031,234.499,-59.097,-176.967,6.123,148.198
C05080=1235.035,234.251,-59.071,-176.970,6.121,148.199
C05081=1235.039,234.002,-59.045,-176.972,6.119,148.199
C05082=1235.044,233.754,-59.020,-176.975,6.117,148.199
C05083=1235.048,233.505,-58.994,-176.977,6.115,148.199
C05084=1235.053,233.256,-58.969,-176.980,6.113,148.200
C05085=1235.057,233.007,-58.944,-176.982,6.111,148.200
C05086=1235.062,232.759,-58.918,-176.985,6.110,148.200
C05087=1235.066,232.510,-58.892,-176.987,6.108,148.201
C05088=1235.071,232.262,-58.867,-176.990,6.107,148.201
C05089=1235.075,232.013,-58.841,-176.992,6.105,148.201
C05090=1235.080,231.764,-58.816,-176.995,6.103,148.202
C05091=1235.084,231.515,-58.791,-176.998,6.101,148.202
C05092=1235.089,231.267,-58.765,-177.000,6.099,148.202
C05093=1235.093,231.018,-58.739,-177.002,6.098,148.203
C05094=1235.098,230.769,-58.714,-177.005,6.096,148.203
C05095=1235.103,230.521,-58.689,-177.007,6.094,148.203
C05096=1235.107,230.272,-58.663,-177.010,6.092,148.204
C05097=1235.111,230.023,-58.637,-177.013,6.090,148.204
C05098=1235.116,229.775,-58.613,-177.015,6.089,148.204
C05099=1235.121,229.526,-58.587,-177.017,6.088,148.205
C05100=1235.125,229.278,-58.562,-177.020,6.086,148.205
C05101=1235.130,229.028,-58.537,-177.023,6.084,148.205
C05102=1235.134,228.779,-58.511,-177.025,6.082,148.206
C05103=1235.139,228.531,-58.485,-177.028,6.080,148.206
C05104=1235.143,228.282,-58.461,-177.031,6.078,148.206
C05105=1235.148,228.034,-58.436,-177.033,6.077,148.207
C05106=1235.152,227.785,-58.410,-177.035,6.075,148.207
C05107=1235.157,227.537,-58.385,-177.038,6.073,148.207
C05108=1235.161,227.288,-58.359,-177.040,6.071,148.208
C05109=1235.166,227.039,-58.335,-177.043,6.070,148.208
C05110=1235.171,226.790,-58.309,-177.046,6.068,148.208
C05111=1235.174,226.542,-58.284,-177.048,6.067,148.209
C05112=1235.179,226.293,-58.259,-177.050,6.065,148.209
C05113=1235.183,226.044,-58.233,-177.053,6.063,148.209
C05114=1235.188,225.796,-58.209,-177.056,6.061,148.210
C05115=1235.193,225.547,-58.183,-177.058,6.059,148.210
C05116=1235.197,225.298,-58.159,-177.061,6.057,148.210
C05117=1235.201,225.050,-58.133,-177.063,6.056,148.211
C05118=1235.206,224.801,-58.109,-177.066,6.054,148.211
C05119=1235.211,224.552,-58.083,-177.068,6.052,148.211
C05120=1235.216,224.303,-58.058,-177.071,6.051,148.212
C05121=1235.219,224.055,-58.033,-177.073,6.049,148.212
C05122=1235.224,223.806,-58.008,-177.075,6.048,148.212
C05123=1235.229,223.557,-57.983,-177.078,6.046,148.213
C05124=1235.234,223.309,-57.958,-177.081,6.044,148.213
C05125=1235.238,223.061,-57.933,-177.083,6.042,148.213
C05126=1235.242,222.811,-57.908,-177.086,6.040,148.214
C05127=1235.248,222.563,-57.883,-177.089,6.038,148.214
C05128=1235.252,222.314,-57.858,-177.091,6.037,148.214
C05129=1235.256,222.065,-57.834,-177.093,6.035,148.215
C05130=1235.260,221.817,-57.808,-177.096,6.034,148.215
C05131=1235.266,221.568,-57.783,-177.098,6.032,148.215
C05132=1235.269,221.319,-57.759,-177.101,6.030,148.215
C05133=1235.274,221.071,-57.733,-177.103,6.029,148.216
C05134=1235.279,220.821,-57.708,-177.106,6.027,148.216
C05135=1235.283,220.573,-57.684,-177.108,6.025,148.217
C05136=1235.288,220.325,-57.659,-177.111,6.023,148.217
C05137=1235.292,220.075,-57.634,-177.114,6.021,148.217
C05138=1235.297,219.827,-57.610,-177.116,6.020,148.218
C05139=1235.301,219.577,-57.585,-177.119,6.019,148.218
C05140=1235.306,219.329,-57.559,-177.121,6.017,148.218
C05141=1235.311,219.081,-57.535,-177.124,6.015,148.219
C05142=1235.315,218.831,-57.510,-177.127,6.013,148.219
C05143=1235.319,218.583,-57.486,-177.129,6.012,148.219
C05144=1235.324,218.334,-57.460,-177.131,6.010,148.220
C05145=1235.329,218.086,-57.436,-177.134,6.008,148.220
C05146=1235.333,217.837,-57.412,-177.137,6.006,148.220
C05147=1235.338,217.588,-57.387,-177.139,6.004,148.221
C05148=1235.342,217.339,-57.363,-177.141,6.003,148.221
C05149=1235.346,217.090,-57.337,-177.144,6.002,148.221
C05150=1235.351,216.842,-57.313,-177.147,6.000,148.222
C05151=1235.356,216.593,-57.288,-177.149,5.998,148.222
C05152=1235.360,216.344,-57.263,-177.152,5.996,148.222
C05153=1235.365,216.095,-57.239,-177.154,5.995,148.223
C05154=1235.370,215.847,-57.214,-177.157,5.993,148.223
C05155=1235.374,215.598,-57.190,-177.160,5.992,148.224
C05156=1235.379,215.350,-57.164,-177.162,5.990,148.224
C05157=1235.383,215.101,-57.140,-177.164,5.989,148.224
C05158=1235.388,214.852,-57.115,-177.167,5.987,148.225
C05159=1235.392,214.603,-57.091,-177.170,5.985,148.225
C05160=1235.397,214.355,-57.067,-177.172,5.983,148.225
C05161=1235.401,214.105,-57.042,-177.175,5.981,148.226
C05162=1235.406,213.857,-57.017,-177.177,5.980,148.226
C05163=1235.410,213.608,-56.993,-177.180,5.978,148.226
C05164=1235.415,213.359,-56.968,-177.183,5.977,148.227
C05165=1235.419,213.110,-56.944,-177.185,5.975,148.227
C05166=1235.424,212.862,-56.920,-177.187,5.974,148.228
C05167=1235.429,212.613,-56.896,-177.190,5.972,148.228
C05168=1235.433,212.364,-56.871,-177.193,5.970,148.228
C05169=1235.438,212.094,-56.844,-177.195,5.968,148.229
C05170=1235.443,211.823,-56.818,-177.198,5.967,148.229
C05171=1235.448,211.553,-56.792,-177.201,5.965,148.230
C05172=1235.453,211.282,-56.765,-177.204,5.963,148.230
C05173=1235.457,211.034,-56.741,-177.206,5.961,148.230
C05174=1235.462,210.785,-56.716,-177.208,5.960,148.231
C05175=1235.467,210.537,-56.692,-177.211,5.958,148.231
C05176=1235.471,210.288,-56.667,-177.214,5.957,148.231
C05177=1235.476,210.038,-56.643,-177.217,5.955,148.232
C05178=1235.480,209.790,-56.619,-177.219,5.954,148.232
C05179=1235.485,209.541,-56.595,-177.221,5.952,148.232
C05180=1235.489,209.292,-56.570,-177.224,5.950,148.233
C05181=1235.494,209.044,-56.546,-177.227,5.948,148.233
C05182=1235.498,208.795,-56.522,-177.229,5.947,148.234
C05183=1235.504,208.546,-56.498,-177.232,5.945,148.234
C05184=1235.508,208.297,-56.474,-177.234,5.944,148.234
C05185=1235.512,208.048,-56.450,-177.237,5.942,148.235
C05186=1235.517,207.800,-56.425,-177.239,5.941,148.235
C05187=1235.521,207.551,-56.401,-177.242,5.939,148.235
C05188=1235.526,207.302,-56.377,-177.244,5.937,148.236
C05189=1235.530,207.054,-56.353,-177.247,5.935,148.236
C05190=1235.535,206.804,-56.328,-177.249,5.934,148.236
C05191=1235.539,206.556,-56.304,-177.252,5.933,148.237
C05192=1235.544,206.307,-56.281,-177.255,5.931,148.237
C05193=1235.549,206.058,-56.256,-177.257,5.930,148.238
C05194=1235.554,205.810,-56.232,-177.260,5.928,148.238
C05195=1235.558,205.560,-56.208,-177.262,5.926,148.238
C05196=1235.562,205.312,-56.184,-177.265,5.924,148.239
C05197=1235.566,205.063,-56.160,-177.267,5.923,148.239
C05198=1235.572,204.814,-56.136,-177.270,5.921,148.240
C05199=1235.576,204.565,-56.112,-177.273,5.920,148.240
C05200=1235.581,204.317,-56.088,-177.275,5.919,148.240
C05201=1235.585,204.068,-56.065,-177.277,5.917,148.241
C05202=1235.589,203.819,-56.040,-177.280,5.915,148.241
C05203=1235.594,203.570,-56.016,-177.283,5.913,148.241
C05204=1235.599,203.321,-55.992,-177.285,5.912,148.242
C05205=1235.603,203.073,-55.968,-177.288,5.910,148.242
C05206=1235.608,202.824,-55.945,-177.290,5.909,148.243
C05207=1235.612,202.575,-55.921,-177.293,5.908,148.243
C05208=1235.618,202.326,-55.897,-177.295,5.906,148.243
C05209=1235.622,202.077,-55.873,-177.298,5.904,148.244
C05210=1235.626,201.828,-55.848,-177.300,5.903,148.244
C05211=1235.631,201.579,-55.825,-177.303,5.901,148.245
C05212=1235.635,201.331,-55.801,-177.306,5.899,148.245
C05213=1235.640,201.082,-55.778,-177.308,5.898,148.245
C05214=1235.644,200.833,-55.754,-177.310,5.896,148.246
C05215=1235.649,200.584,-55.730,-177.313,5.895,148.246
C05216=1235.653,200.336,-55.706,-177.316,5.893,148.247
C05217=1235.659,200.087,-55.682,-177.318,5.892,148.247
C05218=1235.664,199.838,-55.659,-177.321,5.890,148.247
C05219=1235.668,199.589,-55.635,-177.323,5.888,148.248
C05220=1235.673,199.340,-55.611,-177.326,5.887,148.248
C05221=1235.677,199.092,-55.587,-177.329,5.886,148.249
C05222=1235.682,198.843,-55.564,-177.331,5.884,148.249
C05223=1235.686,198.594,-55.539,-177.333,5.883,148.249
C05224=1235.690,198.345,-55.516,-177.336,5.881,148.250
C05225=1235.695,198.096,-55.493,-177.339,5.879,148.250
C05226=1235.699,197.847,-55.469,-177.341,5.878,148.251
C05227=1235.704,197.598,-55.445,-177.344,5.877,148.251
C05228=1235.709,197.349,-55.422,-177.347,5.875,148.251
C05229=1235.713,197.101,-55.398,-177.349,5.874,148.252
C05230=1235.718,196.852,-55.375,-177.351,5.872,148.252
C05231=1235.723,196.603,-55.351,-177.354,5.870,148.253
C05232=1235.727,196.354,-55.327,-177.356,5.869,148.253
C05233=1235.732,196.105,-55.304,-177.359,5.867,148.253
C05234=1235.736,195.856,-55.280,-177.362,5.866,148.254
C05235=1235.741,195.608,-55.256,-177.364,5.865,148.254
C05236=1235.745,195.359,-55.233,-177.367,5.863,148.255
C05237=1235.750,195.110,-55.210,-177.370,5.861,148.255
C05238=1235.755,194.861,-55.186,-177.372,5.860,148.255
C05239=1235.759,194.612,-55.162,-177.374,5.858,148.256
C05240=1235.764,194.363,-55.139,-177.377,5.856,148.256
C05241=1235.769,194.114,-55.115,-177.379,5.856,148.257
C05242=1235.773,193.865,-55.092,-177.382,5.854,148.257
C05243=1235.778,193.616,-55.069,-177.384,5.853,148.257
C05244=1235.782,193.368,-55.045,-177.387,5.851,148.258
C05245=1235.787,193.120,-55.022,-177.390,5.849,148.258
C05246=1235.792,192.871,-54.999,-177.392,5.848,148.259
C05247=1235.796,192.622,-54.976,-177.395,5.847,148.259
C05248=1235.801,192.373,-54.952,-177.397,5.845,148.259
C05249=1235.806,192.124,-54.929,-177.399,5.844,148.260
C05250=1235.810,191.874,-54.905,-177.403,5.842,148.260
C05251=1235.815,191.626,-54.881,-177.405,5.840,148.261
C05252=1235.819,191.377,-54.859,-177.407,5.839,148.261
C05253=1235.824,191.128,-54.835,-177.410,5.837,148.261
C05254=1235.828,190.879,-54.812,-177.412,5.837,148.262
C05255=1235.833,190.630,-54.789,-177.415,5.835,148.262
C05256=1235.838,190.381,-54.765,-177.418,5.833,148.263
C05257=1235.842,190.132,-54.742,-177.420,5.832,148.263
C05258=1235.847,189.884,-54.719,-177.423,5.830,148.264
C05259=1235.852,189.635,-54.696,-177.425,5.829,148.264
C05260=1235.856,189.386,-54.673,-177.428,5.828,148.264
C05261=1235.861,189.137,-54.649,-177.430,5.826,148.265
C05262=1235.866,188.888,-54.626,-177.433,5.825,148.265
C05263=1235.870,188.639,-54.603,-177.436,5.823,148.266
C05264=1235.874,188.390,-54.580,-177.438,5.821,148.266
C05265=1235.879,188.141,-54.557,-177.440,5.820,148.266
C05266=1235.884,187.892,-54.533,-177.443,5.819,148.267
C05267=1235.888,187.644,-54.511,-177.445,5.818,148.267
C05268=1235.893,187.395,-54.487,-177.448,5.816,148.268
C05269=1235.898,187.146,-54.464,-177.451,5.814,148.268
C05270=1235.902,186.897,-54.441,-177.453,5.813,148.269
C05271=1235.906,186.648,-54.418,-177.456,5.812,148.269
C05272=1235.911,186.399,-54.395,-177.458,5.811,148.269
C05273=1235.916,186.130,-54.370,-177.461,5.809,148.270
C05274=1235.922,185.860,-54.345,-177.464,5.807,148.270
C05275=1235.926,185.590,-54.320,-177.466,5.805,148.271
C05276=1235.932,185.321,-54.295,-177.470,5.804,148.271
C05277=1235.936,185.072,-54.272,-177.472,5.803,148.272
C05278=1235.940,184.823,-54.249,-177.474,5.801,148.272
C05279=1235.946,184.575,-54.226,-177.477,5.800,148.272
C05280=1235.951,184.325,-54.203,-177.480,5.798,148.273
C05281=1235.955,184.076,-54.181,-177.482,5.797,148.273
C05282=1235.959,183.827,-54.157,-177.485,5.796,148.274
C05283=1235.963,183.578,-54.134,-177.487,5.794,148.274
C05284=1235.968,183.330,-54.111,-177.489,5.793,148.275
C05285=1235.973,183.080,-54.089,-177.492,5.791,148.275
C05286=1235.977,182.832,-54.066,-177.495,5.790,148.275
C05287=1235.982,182.583,-54.043,-177.497,5.789,148.276
C05288=1235.987,182.334,-54.019,-177.499,5.788,148.276
C05289=1235.992,182.085,-53.998,-177.503,5.786,148.277
C05290=1235.996,181.836,-53.974,-177.505,5.784,148.277
C05291=1236.000,181.587,-53.951,-177.507,5.783,148.278
C05292=1236.005,181.338,-53.928,-177.510,5.781,148.278
C05293=1236.010,181.090,-53.906,-177.513,5.781,148.278
C05294=1236.015,180.841,-53.883,-177.515,5.779,148.279
C05295=1236.019,180.591,-53.860,-177.517,5.778,148.279
C05296=1236.024,180.342,-53.838,-177.520,5.776,148.280
C05297=1236.029,180.094,-53.815,-177.522,5.775,148.280
C05298=1236.033,179.845,-53.792,-177.525,5.773,148.281
C05299=1236.038,179.595,-53.769,-177.528,5.772,148.281
C05300=1236.042,179.347,-53.747,-177.530,5.771,148.281
C05301=1236.047,179.098,-53.724,-177.533,5.769,148.282
C05302=1236.051,178.849,-53.701,-177.535,5.768,148.282
C05303=1236.056,178.600,-53.678,-177.538,5.766,148.283
C05304=1236.061,178.351,-53.656,-177.540,5.765,148.283
C05305=1236.066,178.102,-53.633,-177.543,5.764,148.284
C05306=1236.070,177.853,-53.611,-177.546,5.763,148.284
C05307=1236.075,177.605,-53.588,-177.548,5.761,148.284
C05308=1236.080,177.355,-53.566,-177.550,5.760,148.285
C05309=1236.084,177.106,-53.543,-177.553,5.759,148.285
C05310=1236.089,176.858,-53.521,-177.556,5.757,148.286
C05311=1236.094,176.609,-53.498,-177.558,5.756,148.286
C05312=1236.098,176.359,-53.476,-177.561,5.754,148.287
C05313=1236.103,176.110,-53.452,-177.563,5.753,148.287
C05314=1236.108,175.862,-53.430,-177.566,5.751,148.288
C05315=1236.112,175.613,-53.408,-177.569,5.751,148.288
C05316=1236.117,175.364,-53.385,-177.571,5.749,148.288
C05317=1236.121,175.115,-53.363,-177.573,5.748,148.289
C05318=1236.126,174.866,-53.340,-177.576,5.746,148.289
C05319=1236.131,174.618,-53.318,-177.579,5.745,148.290
C05320=1236.135,174.368,-53.296,-177.581,5.743,148.290
C05321=1236.140,174.119,-53.272,-177.584,5.743,148.291
C05322=1236.145,173.871,-53.251,-177.586,5.741,148.291
C05323=1236.150,173.621,-53.228,-177.589,5.740,148.292
C05324=1236.154,173.372,-53.205,-177.592,5.738,148.292
C05325=1236.158,173.124,-53.183,-177.594,5.737,148.293
C05326=1236.163,172.874,-53.161,-177.596,5.735,148.293
C05327=1236.168,172.626,-53.138,-177.599,5.735,148.293
C05328=1236.172,172.377,-53.116,-177.602,5.733,148.294
C05329=1236.177,172.127,-53.094,-177.604,5.732,148.294
C05330=1236.182,171.879,-53.071,-177.607,5.730,148.295
C05331=1236.186,171.629,-53.049,-177.609,5.729,148.295
C05332=1236.192,171.381,-53.027,-177.612,5.728,148.296
C05333=1236.196,171.132,-53.004,-177.614,5.727,148.296
C05334=1236.200,170.882,-52.982,-177.617,5.725,148.297
C05335=1236.205,170.634,-52.960,-177.619,5.724,148.297
C05336=1236.209,170.385,-52.937,-177.622,5.723,148.298
C05337=1236.214,170.136,-52.915,-177.624,5.722,148.298
C05338=1236.219,169.887,-52.893,-177.627,5.720,148.298
C05339=1236.224,169.638,-52.871,-177.629,5.719,148.299
C05340=1236.228,169.389,-52.848,-177.632,5.717,148.299
C05341=1236.233,169.141,-52.827,-177.635,5.716,148.300
C05342=1236.237,168.891,-52.805,-177.637,5.715,148.300
C05343=1236.242,168.642,-52.782,-177.639,5.714,148.301
C05344=1236.247,168.393,-52.760,-177.643,5.712,148.301
C05345=1236.251,168.144,-52.738,-177.645,5.711,148.302
C05346=1236.256,167.896,-52.716,-177.647,5.709,148.302
C05347=1236.261,167.646,-52.693,-177.650,5.709,148.303
C05348=1236.266,167.397,-52.672,-177.653,5.707,148.303
C05349=1236.270,167.148,-52.649,-177.655,5.706,148.303
C05350=1236.275,166.899,-52.628,-177.658,5.704,148.304
C05351=1236.279,166.650,-52.606,-177.660,5.703,148.304
C05352=1236.284,166.402,-52.583,-177.663,5.702,148.305
C05353=1236.289,166.152,-52.561,-177.665,5.701,148.305
C05354=1236.294,165.904,-52.539,-177.667,5.700,148.306
C05355=1236.298,165.654,-52.517,-177.670,5.698,148.306
C05356=1236.303,165.406,-52.495,-177.672,5.697,148.307
C05357=1236.307,165.156,-52.473,-177.676,5.696,148.307
C05358=1236.312,164.908,-52.452,-177.678,5.695,148.308
C05359=1236.317,164.658,-52.429,-177.680,5.693,148.308
C05360=1236.322,164.409,-52.407,-177.683,5.692,148.309
C05361=1236.326,164.160,-52.385,-177.686,5.690,148.309
C05362=1236.331,163.911,-52.364,-177.688,5.689,148.309
C05363=1236.335,163.662,-52.341,-177.691,5.688,148.310
C05364=1236.340,163.413,-52.320,-177.693,5.687,148.310
C05365=1236.345,163.165,-52.298,-177.695,5.686,148.311
C05366=1236.349,162.915,-52.276,-177.698,5.684,148.311
C05367=1236.354,162.667,-52.254,-177.700,5.683,148.312
C05368=1236.358,162.417,-52.232,-177.703,5.682,148.312
C05369=1236.363,162.169,-52.211,-177.705,5.681,148.313
C05370=1236.368,161.919,-52.188,-177.709,5.679,148.313
C05371=1236.373,161.670,-52.166,-177.711,5.678,148.314
C05372=1236.377,161.421,-52.144,-177.714,5.677,148.314
C05373=1236.382,161.173,-52.123,-177.716,5.676,148.315
C05374=1236.388,160.923,-52.102,-177.718,5.675,148.315
C05375=1236.392,160.674,-52.080,-177.721,5.673,148.316
C05376=1236.397,160.425,-52.058,-177.723,5.672,148.316
C05377=1236.401,160.157,-52.034,-177.726,5.671,148.317
C05378=1236.407,159.887,-52.011,-177.729,5.669,148.317
C05379=1236.411,159.617,-51.987,-177.732,5.668,148.318
C05380=1236.416,159.349,-51.964,-177.735,5.667,148.318
C05381=1236.421,159.100,-51.942,-177.737,5.666,148.319
C05382=1236.426,158.851,-51.921,-177.740,5.664,148.319
C05383=1236.430,158.602,-51.899,-177.742,5.663,148.320
C05384=1236.435,158.353,-51.877,-177.744,5.662,148.320
C05385=1236.439,158.104,-51.855,-177.747,5.661,148.321
C05386=1236.444,157.855,-51.834,-177.750,5.660,148.321
C05387=1236.449,157.606,-51.813,-177.753,5.658,148.322
C05388=1236.454,157.357,-51.791,-177.755,5.657,148.322
C05389=1236.459,157.108,-51.769,-177.757,5.655,148.322
C05390=1236.463,156.859,-51.747,-177.760,5.655,148.323
C05391=1236.468,156.609,-51.726,-177.762,5.654,148.323
C05392=1236.473,156.361,-51.704,-177.765,5.652,148.324
C05393=1236.478,156.112,-51.683,-177.767,5.651,148.324
C05394=1236.482,155.863,-51.661,-177.771,5.650,148.325
C05395=1236.487,155.613,-51.640,-177.773,5.649,148.325
C05396=1236.492,155.365,-51.618,-177.775,5.648,148.326
C05397=1236.496,155.116,-51.597,-177.778,5.646,148.326
C05398=1236.501,154.866,-51.576,-177.780,5.645,148.327
C05399=1236.506,154.618,-51.554,-177.783,5.644,148.327
C05400=1236.510,154.368,-51.532,-177.785,5.643,148.328
C05401=1236.515,154.119,-51.511,-177.788,5.642,148.328
C05402=1236.520,153.871,-51.489,-177.790,5.640,148.329
C05403=1236.525,153.621,-51.468,-177.793,5.640,148.329
C05404=1236.529,153.372,-51.447,-177.796,5.638,148.330
C05405=1236.533,153.124,-51.425,-177.798,5.637,148.330
C05406=1236.539,152.874,-51.404,-177.800,5.636,148.331
C05407=1236.543,152.625,-51.382,-177.804,5.635,148.331
C05408=1236.548,152.376,-51.361,-177.806,5.634,148.332
C05409=1236.553,152.127,-51.339,-177.808,5.633,148.332
C05410=1236.557,151.878,-51.319,-177.811,5.631,148.333
C05411=1236.562,151.629,-51.297,-177.813,5.630,148.333
C05412=1236.567,151.380,-51.275,-177.816,5.629,148.334
C05413=1236.572,151.131,-51.254,-177.818,5.628,148.334
C05414=1236.576,150.883,-51.233,-177.821,5.627,148.335
C05415=1236.580,150.633,-51.212,-177.824,5.625,148.335
C05416=1236.585,150.384,-51.190,-177.826,5.624,148.336
C05417=1236.590,150.135,-51.169,-177.828,5.623,148.336
C05418=1236.595,149.886,-51.148,-177.831,5.622,148.337
C05419=1236.599,149.636,-51.127,-177.833,5.621,148.337
C05420=1236.604,149.387,-51.106,-177.837,5.619,148.338
C05421=1236.609,149.139,-51.084,-177.839,5.618,148.338
C05422=1236.614,148.890,-51.064,-177.841,5.618,148.339
C05423=1236.619,148.641,-51.042,-177.844,5.616,148.339
C05424=1236.623,148.391,-51.021,-177.847,5.615,148.340
C05425=1236.628,148.142,-50.999,-177.849,5.614,148.340
C05426=1236.632,147.893,-50.979,-177.852,5.613,148.341
C05427=1236.638,147.644,-50.958,-177.854,5.612,148.341
C05428=1236.642,147.395,-50.936,-177.857,5.611,148.342
C05429=1236.646,147.146,-50.915,-177.859,5.609,148.342
C05430=1236.651,146.897,-50.894,-177.861,5.608,148.342
C05431=1236.656,146.648,-50.873,-177.864,5.607,148.343
C05432=1236.661,146.399,-50.852,-177.867,5.606,148.343
C05433=1236.666,146.150,-50.831,-177.869,5.605,148.344
C05434=1236.670,145.900,-50.809,-177.872,5.603,148.344
C05435=1236.675,145.651,-50.789,-177.874,5.603,148.345
C05436=1236.680,145.402,-50.768,-177.877,5.602,148.345
C05437=1236.684,145.154,-50.747,-177.880,5.600,148.346
C05438=1236.689,144.905,-50.726,-177.882,5.599,148.346
C05439=1236.694,144.655,-50.705,-177.884,5.599,148.347
C05440=1236.698,144.406,-50.684,-177.887,5.597,148.347
C05441=1236.703,144.157,-50.663,-177.890,5.596,148.348
C05442=1236.707,143.908,-50.642,-177.892,5.595,148.349
C05443=1236.713,143.659,-50.621,-177.895,5.594,148.349
C05444=1236.717,143.410,-50.600,-177.898,5.593,148.350
C05445=1236.722,143.161,-50.579,-177.900,5.592,148.350
C05446=1236.727,142.912,-50.558,-177.903,5.590,148.351
C05447=1236.732,142.663,-50.538,-177.905,5.589,148.351
C05448=1236.736,142.413,-50.516,-177.907,5.589,148.352
C05449=1236.740,142.165,-50.495,-177.910,5.587,148.352
C05450=1236.745,141.916,-50.474,-177.913,5.586,148.353
C05451=1236.751,141.666,-50.453,-177.915,5.585,148.353
C05452=1236.755,141.417,-50.433,-177.918,5.584,148.354
C05453=1236.760,141.168,-50.412,-177.920,5.583,148.354
C05454=1236.765,140.919,-50.392,-177.923,5.582,148.355
C05455=1236.770,140.670,-50.371,-177.925,5.581,148.355
C05456=1236.774,140.422,-50.350,-177.928,5.580,148.356
C05457=1236.779,140.172,-50.329,-177.930,5.579,148.356
C05458=1236.783,139.923,-50.308,-177.933,5.578,148.357
C05459=1236.788,139.673,-50.287,-177.935,5.576,148.357
C05460=1236.793,139.424,-50.267,-177.938,5.576,148.358
C05461=1236.798,139.175,-50.246,-177.940,5.575,148.358
C05462=1236.802,138.926,-50.225,-177.943,5.573,148.359
C05463=1236.807,138.677,-50.205,-177.945,5.572,148.359
C05464=1236.812,138.428,-50.184,-177.948,5.571,148.360
C05465=1236.816,138.179,-50.164,-177.951,5.570,148.361
C05466=1236.821,137.930,-50.143,-177.953,5.569,148.361
